   // GBK_TO_UNICODE[6993] := 16#6436;
   // GBK_TO_UNICODE[6994] := 16#938D;
   // GBK_TO_UNICODE[6995] := 16#6437;
   // GBK_TO_UNICODE[6996] := 16#938E;
   // GBK_TO_UNICODE[6997] := 16#6438;
   // GBK_TO_UNICODE[6998] := 16#938F;
   // GBK_TO_UNICODE[6999] := 16#6439;
   // GBK_TO_UNICODE[7000] := 16#9390;
   // GBK_TO_UNICODE[7001] := 16#643B;
   // GBK_TO_UNICODE[7002] := 16#9391;
   // GBK_TO_UNICODE[7003] := 16#643C;
   // GBK_TO_UNICODE[7004] := 16#9392;
   // GBK_TO_UNICODE[7005] := 16#643E;
   // GBK_TO_UNICODE[7006] := 16#9393;
   // GBK_TO_UNICODE[7007] := 16#6440;
   // GBK_TO_UNICODE[7008] := 16#9394;
   // GBK_TO_UNICODE[7009] := 16#6442;
   // GBK_TO_UNICODE[7010] := 16#9395;
   // GBK_TO_UNICODE[7011] := 16#6443;
   // GBK_TO_UNICODE[7012] := 16#9396;
   // GBK_TO_UNICODE[7013] := 16#6449;
   // GBK_TO_UNICODE[7014] := 16#9397;
   // GBK_TO_UNICODE[7015] := 16#644B;
   // GBK_TO_UNICODE[7016] := 16#9398;
   // GBK_TO_UNICODE[7017] := 16#644C;
   // GBK_TO_UNICODE[7018] := 16#9399;
   // GBK_TO_UNICODE[7019] := 16#644D;
   // GBK_TO_UNICODE[7020] := 16#939A;
   // GBK_TO_UNICODE[7021] := 16#644E;
   // GBK_TO_UNICODE[7022] := 16#939B;
   // GBK_TO_UNICODE[7023] := 16#644F;
   // GBK_TO_UNICODE[7024] := 16#939C;
   // GBK_TO_UNICODE[7025] := 16#6450;
   // GBK_TO_UNICODE[7026] := 16#939D;
   // GBK_TO_UNICODE[7027] := 16#6451;
   // GBK_TO_UNICODE[7028] := 16#939E;
   // GBK_TO_UNICODE[7029] := 16#6453;
   // GBK_TO_UNICODE[7030] := 16#939F;
   // GBK_TO_UNICODE[7031] := 16#6455;
   // GBK_TO_UNICODE[7032] := 16#93A0;
   // GBK_TO_UNICODE[7033] := 16#6456;
   // GBK_TO_UNICODE[7034] := 16#93A1;
   // GBK_TO_UNICODE[7035] := 16#6457;
   // GBK_TO_UNICODE[7036] := 16#93A2;
   // GBK_TO_UNICODE[7037] := 16#6459;
   // GBK_TO_UNICODE[7038] := 16#93A3;
   // GBK_TO_UNICODE[7039] := 16#645A;
   // GBK_TO_UNICODE[7040] := 16#93A4;
   // GBK_TO_UNICODE[7041] := 16#645B;
   // GBK_TO_UNICODE[7042] := 16#93A5;
   // GBK_TO_UNICODE[7043] := 16#645C;
   // GBK_TO_UNICODE[7044] := 16#93A6;
   // GBK_TO_UNICODE[7045] := 16#645D;
   // GBK_TO_UNICODE[7046] := 16#93A7;
   // GBK_TO_UNICODE[7047] := 16#645F;
   // GBK_TO_UNICODE[7048] := 16#93A8;
   // GBK_TO_UNICODE[7049] := 16#6460;
   // GBK_TO_UNICODE[7050] := 16#93A9;
   // GBK_TO_UNICODE[7051] := 16#6461;
   // GBK_TO_UNICODE[7052] := 16#93AA;
   // GBK_TO_UNICODE[7053] := 16#6462;
   // GBK_TO_UNICODE[7054] := 16#93AB;
   // GBK_TO_UNICODE[7055] := 16#6463;
   // GBK_TO_UNICODE[7056] := 16#93AC;
   // GBK_TO_UNICODE[7057] := 16#6464;
   // GBK_TO_UNICODE[7058] := 16#93AD;
   // GBK_TO_UNICODE[7059] := 16#6465;
   // GBK_TO_UNICODE[7060] := 16#93AE;
   // GBK_TO_UNICODE[7061] := 16#6466;
   // GBK_TO_UNICODE[7062] := 16#93AF;
   // GBK_TO_UNICODE[7063] := 16#6468;
   // GBK_TO_UNICODE[7064] := 16#93B0;
   // GBK_TO_UNICODE[7065] := 16#646A;
   // GBK_TO_UNICODE[7066] := 16#93B1;
   // GBK_TO_UNICODE[7067] := 16#646B;
   // GBK_TO_UNICODE[7068] := 16#93B2;
   // GBK_TO_UNICODE[7069] := 16#646C;
   // GBK_TO_UNICODE[7070] := 16#93B3;
   // GBK_TO_UNICODE[7071] := 16#646E;
   // GBK_TO_UNICODE[7072] := 16#93B4;
   // GBK_TO_UNICODE[7073] := 16#646F;
   // GBK_TO_UNICODE[7074] := 16#93B5;
   // GBK_TO_UNICODE[7075] := 16#6470;
   // GBK_TO_UNICODE[7076] := 16#93B6;
   // GBK_TO_UNICODE[7077] := 16#6471;
   // GBK_TO_UNICODE[7078] := 16#93B7;
   // GBK_TO_UNICODE[7079] := 16#6472;
   // GBK_TO_UNICODE[7080] := 16#93B8;
   // GBK_TO_UNICODE[7081] := 16#6473;
   // GBK_TO_UNICODE[7082] := 16#93B9;
   // GBK_TO_UNICODE[7083] := 16#6474;
   // GBK_TO_UNICODE[7084] := 16#93BA;
   // GBK_TO_UNICODE[7085] := 16#6475;
   // GBK_TO_UNICODE[7086] := 16#93BB;
   // GBK_TO_UNICODE[7087] := 16#6476;
   // GBK_TO_UNICODE[7088] := 16#93BC;
   // GBK_TO_UNICODE[7089] := 16#6477;
   // GBK_TO_UNICODE[7090] := 16#93BD;
   // GBK_TO_UNICODE[7091] := 16#647B;
   // GBK_TO_UNICODE[7092] := 16#93BE;
   // GBK_TO_UNICODE[7093] := 16#647C;
   // GBK_TO_UNICODE[7094] := 16#93BF;
   // GBK_TO_UNICODE[7095] := 16#647D;
   // GBK_TO_UNICODE[7096] := 16#93C0;
   // GBK_TO_UNICODE[7097] := 16#647E;
   // GBK_TO_UNICODE[7098] := 16#93C1;
   // GBK_TO_UNICODE[7099] := 16#647F;
   // GBK_TO_UNICODE[7100] := 16#93C2;
   // GBK_TO_UNICODE[7101] := 16#6480;
   // GBK_TO_UNICODE[7102] := 16#93C3;
   // GBK_TO_UNICODE[7103] := 16#6481;
   // GBK_TO_UNICODE[7104] := 16#93C4;
   // GBK_TO_UNICODE[7105] := 16#6483;
   // GBK_TO_UNICODE[7106] := 16#93C5;
   // GBK_TO_UNICODE[7107] := 16#6486;
   // GBK_TO_UNICODE[7108] := 16#93C6;
   // GBK_TO_UNICODE[7109] := 16#6488;
   // GBK_TO_UNICODE[7110] := 16#93C7;
   // GBK_TO_UNICODE[7111] := 16#6489;
   // GBK_TO_UNICODE[7112] := 16#93C8;
   // GBK_TO_UNICODE[7113] := 16#648A;
   // GBK_TO_UNICODE[7114] := 16#93C9;
   // GBK_TO_UNICODE[7115] := 16#648B;
   // GBK_TO_UNICODE[7116] := 16#93CA;
   // GBK_TO_UNICODE[7117] := 16#648C;
   // GBK_TO_UNICODE[7118] := 16#93CB;
   // GBK_TO_UNICODE[7119] := 16#648D;
   // GBK_TO_UNICODE[7120] := 16#93CC;
   // GBK_TO_UNICODE[7121] := 16#648E;
   // GBK_TO_UNICODE[7122] := 16#93CD;
   // GBK_TO_UNICODE[7123] := 16#648F;
   // GBK_TO_UNICODE[7124] := 16#93CE;
   // GBK_TO_UNICODE[7125] := 16#6490;
   // GBK_TO_UNICODE[7126] := 16#93CF;
   // GBK_TO_UNICODE[7127] := 16#6493;
   // GBK_TO_UNICODE[7128] := 16#93D0;
   // GBK_TO_UNICODE[7129] := 16#6494;
   // GBK_TO_UNICODE[7130] := 16#93D1;
   // GBK_TO_UNICODE[7131] := 16#6497;
   // GBK_TO_UNICODE[7132] := 16#93D2;
   // GBK_TO_UNICODE[7133] := 16#6498;
   // GBK_TO_UNICODE[7134] := 16#93D3;
   // GBK_TO_UNICODE[7135] := 16#649A;
   // GBK_TO_UNICODE[7136] := 16#93D4;
   // GBK_TO_UNICODE[7137] := 16#649B;
   // GBK_TO_UNICODE[7138] := 16#93D5;
   // GBK_TO_UNICODE[7139] := 16#649C;
   // GBK_TO_UNICODE[7140] := 16#93D6;
   // GBK_TO_UNICODE[7141] := 16#649D;
   // GBK_TO_UNICODE[7142] := 16#93D7;
   // GBK_TO_UNICODE[7143] := 16#649F;
   // GBK_TO_UNICODE[7144] := 16#93D8;
   // GBK_TO_UNICODE[7145] := 16#64A0;
   // GBK_TO_UNICODE[7146] := 16#93D9;
   // GBK_TO_UNICODE[7147] := 16#64A1;
   // GBK_TO_UNICODE[7148] := 16#93DA;
   // GBK_TO_UNICODE[7149] := 16#64A2;
   // GBK_TO_UNICODE[7150] := 16#93DB;
   // GBK_TO_UNICODE[7151] := 16#64A3;
   // GBK_TO_UNICODE[7152] := 16#93DC;
   // GBK_TO_UNICODE[7153] := 16#64A5;
   // GBK_TO_UNICODE[7154] := 16#93DD;
   // GBK_TO_UNICODE[7155] := 16#64A6;
   // GBK_TO_UNICODE[7156] := 16#93DE;
   // GBK_TO_UNICODE[7157] := 16#64A7;
   // GBK_TO_UNICODE[7158] := 16#93DF;
   // GBK_TO_UNICODE[7159] := 16#64A8;
   // GBK_TO_UNICODE[7160] := 16#93E0;
   // GBK_TO_UNICODE[7161] := 16#64AA;
   // GBK_TO_UNICODE[7162] := 16#93E1;
   // GBK_TO_UNICODE[7163] := 16#64AB;
   // GBK_TO_UNICODE[7164] := 16#93E2;
   // GBK_TO_UNICODE[7165] := 16#64AF;
   // GBK_TO_UNICODE[7166] := 16#93E3;
   // GBK_TO_UNICODE[7167] := 16#64B1;
   // GBK_TO_UNICODE[7168] := 16#93E4;
   // GBK_TO_UNICODE[7169] := 16#64B2;
   // GBK_TO_UNICODE[7170] := 16#93E5;
   // GBK_TO_UNICODE[7171] := 16#64B3;
   // GBK_TO_UNICODE[7172] := 16#93E6;
   // GBK_TO_UNICODE[7173] := 16#64B4;
   // GBK_TO_UNICODE[7174] := 16#93E7;
   // GBK_TO_UNICODE[7175] := 16#64B6;
   // GBK_TO_UNICODE[7176] := 16#93E8;
   // GBK_TO_UNICODE[7177] := 16#64B9;
   // GBK_TO_UNICODE[7178] := 16#93E9;
   // GBK_TO_UNICODE[7179] := 16#64BB;
   // GBK_TO_UNICODE[7180] := 16#93EA;
   // GBK_TO_UNICODE[7181] := 16#64BD;
   // GBK_TO_UNICODE[7182] := 16#93EB;
   // GBK_TO_UNICODE[7183] := 16#64BE;
   // GBK_TO_UNICODE[7184] := 16#93EC;
   // GBK_TO_UNICODE[7185] := 16#64BF;
   // GBK_TO_UNICODE[7186] := 16#93ED;
   // GBK_TO_UNICODE[7187] := 16#64C1;
   // GBK_TO_UNICODE[7188] := 16#93EE;
   // GBK_TO_UNICODE[7189] := 16#64C3;
   // GBK_TO_UNICODE[7190] := 16#93EF;
   // GBK_TO_UNICODE[7191] := 16#64C4;
   // GBK_TO_UNICODE[7192] := 16#93F0;
   // GBK_TO_UNICODE[7193] := 16#64C6;
   // GBK_TO_UNICODE[7194] := 16#93F1;
   // GBK_TO_UNICODE[7195] := 16#64C7;
   // GBK_TO_UNICODE[7196] := 16#93F2;
   // GBK_TO_UNICODE[7197] := 16#64C8;
   // GBK_TO_UNICODE[7198] := 16#93F3;
   // GBK_TO_UNICODE[7199] := 16#64C9;
   // GBK_TO_UNICODE[7200] := 16#93F4;
   // GBK_TO_UNICODE[7201] := 16#64CA;
   // GBK_TO_UNICODE[7202] := 16#93F5;
   // GBK_TO_UNICODE[7203] := 16#64CB;
   // GBK_TO_UNICODE[7204] := 16#93F6;
   // GBK_TO_UNICODE[7205] := 16#64CC;
   // GBK_TO_UNICODE[7206] := 16#93F7;
   // GBK_TO_UNICODE[7207] := 16#64CF;
   // GBK_TO_UNICODE[7208] := 16#93F8;
   // GBK_TO_UNICODE[7209] := 16#64D1;
   // GBK_TO_UNICODE[7210] := 16#93F9;
   // GBK_TO_UNICODE[7211] := 16#64D3;
   // GBK_TO_UNICODE[7212] := 16#93FA;
   // GBK_TO_UNICODE[7213] := 16#64D4;
   // GBK_TO_UNICODE[7214] := 16#93FB;
   // GBK_TO_UNICODE[7215] := 16#64D5;
   // GBK_TO_UNICODE[7216] := 16#93FC;
   // GBK_TO_UNICODE[7217] := 16#64D6;
   // GBK_TO_UNICODE[7218] := 16#93FD;
   // GBK_TO_UNICODE[7219] := 16#64D9;
   // GBK_TO_UNICODE[7220] := 16#93FE;
   // GBK_TO_UNICODE[7221] := 16#64DA;
   // GBK_TO_UNICODE[7222] := 16#9440;
   // GBK_TO_UNICODE[7223] := 16#64DB;
   // GBK_TO_UNICODE[7224] := 16#9441;
   // GBK_TO_UNICODE[7225] := 16#64DC;
   // GBK_TO_UNICODE[7226] := 16#9442;
   // GBK_TO_UNICODE[7227] := 16#64DD;
   // GBK_TO_UNICODE[7228] := 16#9443;
   // GBK_TO_UNICODE[7229] := 16#64DF;
   // GBK_TO_UNICODE[7230] := 16#9444;
   // GBK_TO_UNICODE[7231] := 16#64E0;
   // GBK_TO_UNICODE[7232] := 16#9445;
   // GBK_TO_UNICODE[7233] := 16#64E1;
   // GBK_TO_UNICODE[7234] := 16#9446;
   // GBK_TO_UNICODE[7235] := 16#64E3;
   // GBK_TO_UNICODE[7236] := 16#9447;
   // GBK_TO_UNICODE[7237] := 16#64E5;
   // GBK_TO_UNICODE[7238] := 16#9448;
   // GBK_TO_UNICODE[7239] := 16#64E7;
   // GBK_TO_UNICODE[7240] := 16#9449;
   // GBK_TO_UNICODE[7241] := 16#64E8;
   // GBK_TO_UNICODE[7242] := 16#944A;
   // GBK_TO_UNICODE[7243] := 16#64E9;
   // GBK_TO_UNICODE[7244] := 16#944B;
   // GBK_TO_UNICODE[7245] := 16#64EA;
   // GBK_TO_UNICODE[7246] := 16#944C;
   // GBK_TO_UNICODE[7247] := 16#64EB;
   // GBK_TO_UNICODE[7248] := 16#944D;
   // GBK_TO_UNICODE[7249] := 16#64EC;
   // GBK_TO_UNICODE[7250] := 16#944E;
   // GBK_TO_UNICODE[7251] := 16#64ED;
   // GBK_TO_UNICODE[7252] := 16#944F;
   // GBK_TO_UNICODE[7253] := 16#64EE;
   // GBK_TO_UNICODE[7254] := 16#9450;
   // GBK_TO_UNICODE[7255] := 16#64EF;
   // GBK_TO_UNICODE[7256] := 16#9451;
   // GBK_TO_UNICODE[7257] := 16#64F0;
   // GBK_TO_UNICODE[7258] := 16#9452;
   // GBK_TO_UNICODE[7259] := 16#64F1;
   // GBK_TO_UNICODE[7260] := 16#9453;
   // GBK_TO_UNICODE[7261] := 16#64F2;
   // GBK_TO_UNICODE[7262] := 16#9454;
   // GBK_TO_UNICODE[7263] := 16#64F3;
   // GBK_TO_UNICODE[7264] := 16#9455;
   // GBK_TO_UNICODE[7265] := 16#64F4;
   // GBK_TO_UNICODE[7266] := 16#9456;
   // GBK_TO_UNICODE[7267] := 16#64F5;
   // GBK_TO_UNICODE[7268] := 16#9457;
   // GBK_TO_UNICODE[7269] := 16#64F6;
   // GBK_TO_UNICODE[7270] := 16#9458;
   // GBK_TO_UNICODE[7271] := 16#64F7;
   // GBK_TO_UNICODE[7272] := 16#9459;
   // GBK_TO_UNICODE[7273] := 16#64F8;
   // GBK_TO_UNICODE[7274] := 16#945A;
   // GBK_TO_UNICODE[7275] := 16#64F9;
   // GBK_TO_UNICODE[7276] := 16#945B;
   // GBK_TO_UNICODE[7277] := 16#64FA;
   // GBK_TO_UNICODE[7278] := 16#945C;
   // GBK_TO_UNICODE[7279] := 16#64FB;
   // GBK_TO_UNICODE[7280] := 16#945D;
   // GBK_TO_UNICODE[7281] := 16#64FC;
   // GBK_TO_UNICODE[7282] := 16#945E;
   // GBK_TO_UNICODE[7283] := 16#64FD;
   // GBK_TO_UNICODE[7284] := 16#945F;
   // GBK_TO_UNICODE[7285] := 16#64FE;
   // GBK_TO_UNICODE[7286] := 16#9460;
   // GBK_TO_UNICODE[7287] := 16#64FF;
   // GBK_TO_UNICODE[7288] := 16#9461;
   // GBK_TO_UNICODE[7289] := 16#6501;
   // GBK_TO_UNICODE[7290] := 16#9462;
   // GBK_TO_UNICODE[7291] := 16#6502;
   // GBK_TO_UNICODE[7292] := 16#9463;
   // GBK_TO_UNICODE[7293] := 16#6503;
   // GBK_TO_UNICODE[7294] := 16#9464;
   // GBK_TO_UNICODE[7295] := 16#6504;
   // GBK_TO_UNICODE[7296] := 16#9465;
   // GBK_TO_UNICODE[7297] := 16#6505;
   // GBK_TO_UNICODE[7298] := 16#9466;
   // GBK_TO_UNICODE[7299] := 16#6506;
   // GBK_TO_UNICODE[7300] := 16#9467;
   // GBK_TO_UNICODE[7301] := 16#6507;
   // GBK_TO_UNICODE[7302] := 16#9468;
   // GBK_TO_UNICODE[7303] := 16#6508;
   // GBK_TO_UNICODE[7304] := 16#9469;
   // GBK_TO_UNICODE[7305] := 16#650A;
   // GBK_TO_UNICODE[7306] := 16#946A;
   // GBK_TO_UNICODE[7307] := 16#650B;
   // GBK_TO_UNICODE[7308] := 16#946B;
   // GBK_TO_UNICODE[7309] := 16#650C;
   // GBK_TO_UNICODE[7310] := 16#946C;
   // GBK_TO_UNICODE[7311] := 16#650D;
   // GBK_TO_UNICODE[7312] := 16#946D;
   // GBK_TO_UNICODE[7313] := 16#650E;
   // GBK_TO_UNICODE[7314] := 16#946E;
   // GBK_TO_UNICODE[7315] := 16#650F;
   // GBK_TO_UNICODE[7316] := 16#946F;
   // GBK_TO_UNICODE[7317] := 16#6510;
   // GBK_TO_UNICODE[7318] := 16#9470;
   // GBK_TO_UNICODE[7319] := 16#6511;
   // GBK_TO_UNICODE[7320] := 16#9471;
   // GBK_TO_UNICODE[7321] := 16#6513;
   // GBK_TO_UNICODE[7322] := 16#9472;
   // GBK_TO_UNICODE[7323] := 16#6514;
   // GBK_TO_UNICODE[7324] := 16#9473;
   // GBK_TO_UNICODE[7325] := 16#6515;
   // GBK_TO_UNICODE[7326] := 16#9474;
   // GBK_TO_UNICODE[7327] := 16#6516;
   // GBK_TO_UNICODE[7328] := 16#9475;
   // GBK_TO_UNICODE[7329] := 16#6517;
   // GBK_TO_UNICODE[7330] := 16#9476;
   // GBK_TO_UNICODE[7331] := 16#6519;
   // GBK_TO_UNICODE[7332] := 16#9477;
   // GBK_TO_UNICODE[7333] := 16#651A;
   // GBK_TO_UNICODE[7334] := 16#9478;
   // GBK_TO_UNICODE[7335] := 16#651B;
   // GBK_TO_UNICODE[7336] := 16#9479;
   // GBK_TO_UNICODE[7337] := 16#651C;
   // GBK_TO_UNICODE[7338] := 16#947A;
   // GBK_TO_UNICODE[7339] := 16#651D;
   // GBK_TO_UNICODE[7340] := 16#947B;
   // GBK_TO_UNICODE[7341] := 16#651E;
   // GBK_TO_UNICODE[7342] := 16#947C;
   // GBK_TO_UNICODE[7343] := 16#651F;
   // GBK_TO_UNICODE[7344] := 16#947D;
   // GBK_TO_UNICODE[7345] := 16#6520;
   // GBK_TO_UNICODE[7346] := 16#947E;
   // GBK_TO_UNICODE[7347] := 16#6521;
   // GBK_TO_UNICODE[7348] := 16#9480;
   // GBK_TO_UNICODE[7349] := 16#6522;
   // GBK_TO_UNICODE[7350] := 16#9481;
   // GBK_TO_UNICODE[7351] := 16#6523;
   // GBK_TO_UNICODE[7352] := 16#9482;
   // GBK_TO_UNICODE[7353] := 16#6524;
   // GBK_TO_UNICODE[7354] := 16#9483;
   // GBK_TO_UNICODE[7355] := 16#6526;
   // GBK_TO_UNICODE[7356] := 16#9484;
   // GBK_TO_UNICODE[7357] := 16#6527;
   // GBK_TO_UNICODE[7358] := 16#9485;
   // GBK_TO_UNICODE[7359] := 16#6528;
   // GBK_TO_UNICODE[7360] := 16#9486;
   // GBK_TO_UNICODE[7361] := 16#6529;
   // GBK_TO_UNICODE[7362] := 16#9487;
   // GBK_TO_UNICODE[7363] := 16#652A;
   // GBK_TO_UNICODE[7364] := 16#9488;
   // GBK_TO_UNICODE[7365] := 16#652C;
   // GBK_TO_UNICODE[7366] := 16#9489;
   // GBK_TO_UNICODE[7367] := 16#652D;
   // GBK_TO_UNICODE[7368] := 16#948A;
   // GBK_TO_UNICODE[7369] := 16#6530;
   // GBK_TO_UNICODE[7370] := 16#948B;
   // GBK_TO_UNICODE[7371] := 16#6531;
   // GBK_TO_UNICODE[7372] := 16#948C;
   // GBK_TO_UNICODE[7373] := 16#6532;
   // GBK_TO_UNICODE[7374] := 16#948D;
   // GBK_TO_UNICODE[7375] := 16#6533;
   // GBK_TO_UNICODE[7376] := 16#948E;
   // GBK_TO_UNICODE[7377] := 16#6537;
   // GBK_TO_UNICODE[7378] := 16#948F;
   // GBK_TO_UNICODE[7379] := 16#653A;
   // GBK_TO_UNICODE[7380] := 16#9490;
   // GBK_TO_UNICODE[7381] := 16#653C;
   // GBK_TO_UNICODE[7382] := 16#9491;
   // GBK_TO_UNICODE[7383] := 16#653D;
   // GBK_TO_UNICODE[7384] := 16#9492;
   // GBK_TO_UNICODE[7385] := 16#6540;
   // GBK_TO_UNICODE[7386] := 16#9493;
   // GBK_TO_UNICODE[7387] := 16#6541;
   // GBK_TO_UNICODE[7388] := 16#9494;
   // GBK_TO_UNICODE[7389] := 16#6542;
   // GBK_TO_UNICODE[7390] := 16#9495;
   // GBK_TO_UNICODE[7391] := 16#6543;
   // GBK_TO_UNICODE[7392] := 16#9496;
   // GBK_TO_UNICODE[7393] := 16#6544;
   // GBK_TO_UNICODE[7394] := 16#9497;
   // GBK_TO_UNICODE[7395] := 16#6546;
   // GBK_TO_UNICODE[7396] := 16#9498;
   // GBK_TO_UNICODE[7397] := 16#6547;
   // GBK_TO_UNICODE[7398] := 16#9499;
   // GBK_TO_UNICODE[7399] := 16#654A;
   // GBK_TO_UNICODE[7400] := 16#949A;
   // GBK_TO_UNICODE[7401] := 16#654B;
   // GBK_TO_UNICODE[7402] := 16#949B;
   // GBK_TO_UNICODE[7403] := 16#654D;
   // GBK_TO_UNICODE[7404] := 16#949C;
   // GBK_TO_UNICODE[7405] := 16#654E;
   // GBK_TO_UNICODE[7406] := 16#949D;
   // GBK_TO_UNICODE[7407] := 16#6550;
   // GBK_TO_UNICODE[7408] := 16#949E;
   // GBK_TO_UNICODE[7409] := 16#6552;
   // GBK_TO_UNICODE[7410] := 16#949F;
   // GBK_TO_UNICODE[7411] := 16#6553;
   // GBK_TO_UNICODE[7412] := 16#94A0;
   // GBK_TO_UNICODE[7413] := 16#6554;
   // GBK_TO_UNICODE[7414] := 16#94A1;
   // GBK_TO_UNICODE[7415] := 16#6557;
   // GBK_TO_UNICODE[7416] := 16#94A2;
   // GBK_TO_UNICODE[7417] := 16#6558;
   // GBK_TO_UNICODE[7418] := 16#94A3;
   // GBK_TO_UNICODE[7419] := 16#655A;
   // GBK_TO_UNICODE[7420] := 16#94A4;
   // GBK_TO_UNICODE[7421] := 16#655C;
   // GBK_TO_UNICODE[7422] := 16#94A5;
   // GBK_TO_UNICODE[7423] := 16#655F;
   // GBK_TO_UNICODE[7424] := 16#94A6;
   // GBK_TO_UNICODE[7425] := 16#6560;
   // GBK_TO_UNICODE[7426] := 16#94A7;
   // GBK_TO_UNICODE[7427] := 16#6561;
   // GBK_TO_UNICODE[7428] := 16#94A8;
   // GBK_TO_UNICODE[7429] := 16#6564;
   // GBK_TO_UNICODE[7430] := 16#94A9;
   // GBK_TO_UNICODE[7431] := 16#6565;
   // GBK_TO_UNICODE[7432] := 16#94AA;
   // GBK_TO_UNICODE[7433] := 16#6567;
   // GBK_TO_UNICODE[7434] := 16#94AB;
   // GBK_TO_UNICODE[7435] := 16#6568;
   // GBK_TO_UNICODE[7436] := 16#94AC;
   // GBK_TO_UNICODE[7437] := 16#6569;
   // GBK_TO_UNICODE[7438] := 16#94AD;
   // GBK_TO_UNICODE[7439] := 16#656A;
   // GBK_TO_UNICODE[7440] := 16#94AE;
   // GBK_TO_UNICODE[7441] := 16#656D;
   // GBK_TO_UNICODE[7442] := 16#94AF;
   // GBK_TO_UNICODE[7443] := 16#656E;
   // GBK_TO_UNICODE[7444] := 16#94B0;
   // GBK_TO_UNICODE[7445] := 16#656F;
   // GBK_TO_UNICODE[7446] := 16#94B1;
   // GBK_TO_UNICODE[7447] := 16#6571;
   // GBK_TO_UNICODE[7448] := 16#94B2;
   // GBK_TO_UNICODE[7449] := 16#6573;
   // GBK_TO_UNICODE[7450] := 16#94B3;
   // GBK_TO_UNICODE[7451] := 16#6575;
   // GBK_TO_UNICODE[7452] := 16#94B4;
   // GBK_TO_UNICODE[7453] := 16#6576;
   // GBK_TO_UNICODE[7454] := 16#94B5;
   // GBK_TO_UNICODE[7455] := 16#6578;
   // GBK_TO_UNICODE[7456] := 16#94B6;
   // GBK_TO_UNICODE[7457] := 16#6579;
   // GBK_TO_UNICODE[7458] := 16#94B7;
   // GBK_TO_UNICODE[7459] := 16#657A;
   // GBK_TO_UNICODE[7460] := 16#94B8;
   // GBK_TO_UNICODE[7461] := 16#657B;
   // GBK_TO_UNICODE[7462] := 16#94B9;
   // GBK_TO_UNICODE[7463] := 16#657C;
   // GBK_TO_UNICODE[7464] := 16#94BA;
   // GBK_TO_UNICODE[7465] := 16#657D;
   // GBK_TO_UNICODE[7466] := 16#94BB;
   // GBK_TO_UNICODE[7467] := 16#657E;
   // GBK_TO_UNICODE[7468] := 16#94BC;
   // GBK_TO_UNICODE[7469] := 16#657F;
   // GBK_TO_UNICODE[7470] := 16#94BD;
   // GBK_TO_UNICODE[7471] := 16#6580;
   // GBK_TO_UNICODE[7472] := 16#94BE;
   // GBK_TO_UNICODE[7473] := 16#6581;
   // GBK_TO_UNICODE[7474] := 16#94BF;
   // GBK_TO_UNICODE[7475] := 16#6582;
   // GBK_TO_UNICODE[7476] := 16#94C0;
   // GBK_TO_UNICODE[7477] := 16#6583;
   // GBK_TO_UNICODE[7478] := 16#94C1;
   // GBK_TO_UNICODE[7479] := 16#6584;
   // GBK_TO_UNICODE[7480] := 16#94C2;
   // GBK_TO_UNICODE[7481] := 16#6585;
   // GBK_TO_UNICODE[7482] := 16#94C3;
   // GBK_TO_UNICODE[7483] := 16#6586;
   // GBK_TO_UNICODE[7484] := 16#94C4;
   // GBK_TO_UNICODE[7485] := 16#6588;
   // GBK_TO_UNICODE[7486] := 16#94C5;
   // GBK_TO_UNICODE[7487] := 16#6589;
   // GBK_TO_UNICODE[7488] := 16#94C6;
   // GBK_TO_UNICODE[7489] := 16#658A;
   // GBK_TO_UNICODE[7490] := 16#94C7;
   // GBK_TO_UNICODE[7491] := 16#658D;
   // GBK_TO_UNICODE[7492] := 16#94C8;
   // GBK_TO_UNICODE[7493] := 16#658E;
   // GBK_TO_UNICODE[7494] := 16#94C9;
   // GBK_TO_UNICODE[7495] := 16#658F;
   // GBK_TO_UNICODE[7496] := 16#94CA;
   // GBK_TO_UNICODE[7497] := 16#6592;
   // GBK_TO_UNICODE[7498] := 16#94CB;
   // GBK_TO_UNICODE[7499] := 16#6594;
   // GBK_TO_UNICODE[7500] := 16#94CC;
   // GBK_TO_UNICODE[7501] := 16#6595;
   // GBK_TO_UNICODE[7502] := 16#94CD;
   // GBK_TO_UNICODE[7503] := 16#6596;
   // GBK_TO_UNICODE[7504] := 16#94CE;
   // GBK_TO_UNICODE[7505] := 16#6598;
   // GBK_TO_UNICODE[7506] := 16#94CF;
   // GBK_TO_UNICODE[7507] := 16#659A;
   // GBK_TO_UNICODE[7508] := 16#94D0;
   // GBK_TO_UNICODE[7509] := 16#659D;
   // GBK_TO_UNICODE[7510] := 16#94D1;
   // GBK_TO_UNICODE[7511] := 16#659E;
   // GBK_TO_UNICODE[7512] := 16#94D2;
   // GBK_TO_UNICODE[7513] := 16#65A0;
   // GBK_TO_UNICODE[7514] := 16#94D3;
   // GBK_TO_UNICODE[7515] := 16#65A2;
   // GBK_TO_UNICODE[7516] := 16#94D4;
   // GBK_TO_UNICODE[7517] := 16#65A3;
   // GBK_TO_UNICODE[7518] := 16#94D5;
   // GBK_TO_UNICODE[7519] := 16#65A6;
   // GBK_TO_UNICODE[7520] := 16#94D6;
   // GBK_TO_UNICODE[7521] := 16#65A8;
   // GBK_TO_UNICODE[7522] := 16#94D7;
   // GBK_TO_UNICODE[7523] := 16#65AA;
   // GBK_TO_UNICODE[7524] := 16#94D8;
   // GBK_TO_UNICODE[7525] := 16#65AC;
   // GBK_TO_UNICODE[7526] := 16#94D9;
   // GBK_TO_UNICODE[7527] := 16#65AE;
   // GBK_TO_UNICODE[7528] := 16#94DA;
   // GBK_TO_UNICODE[7529] := 16#65B1;
   // GBK_TO_UNICODE[7530] := 16#94DB;
   // GBK_TO_UNICODE[7531] := 16#65B2;
   // GBK_TO_UNICODE[7532] := 16#94DC;
   // GBK_TO_UNICODE[7533] := 16#65B3;
   // GBK_TO_UNICODE[7534] := 16#94DD;
   // GBK_TO_UNICODE[7535] := 16#65B4;
   // GBK_TO_UNICODE[7536] := 16#94DE;
   // GBK_TO_UNICODE[7537] := 16#65B5;
   // GBK_TO_UNICODE[7538] := 16#94DF;
   // GBK_TO_UNICODE[7539] := 16#65B6;
   // GBK_TO_UNICODE[7540] := 16#94E0;
   // GBK_TO_UNICODE[7541] := 16#65B7;
   // GBK_TO_UNICODE[7542] := 16#94E1;
   // GBK_TO_UNICODE[7543] := 16#65B8;
   // GBK_TO_UNICODE[7544] := 16#94E2;
   // GBK_TO_UNICODE[7545] := 16#65BA;
   // GBK_TO_UNICODE[7546] := 16#94E3;
   // GBK_TO_UNICODE[7547] := 16#65BB;
   // GBK_TO_UNICODE[7548] := 16#94E4;
   // GBK_TO_UNICODE[7549] := 16#65BE;
   // GBK_TO_UNICODE[7550] := 16#94E5;
   // GBK_TO_UNICODE[7551] := 16#65BF;
   // GBK_TO_UNICODE[7552] := 16#94E6;
   // GBK_TO_UNICODE[7553] := 16#65C0;
   // GBK_TO_UNICODE[7554] := 16#94E7;
   // GBK_TO_UNICODE[7555] := 16#65C2;
   // GBK_TO_UNICODE[7556] := 16#94E8;
   // GBK_TO_UNICODE[7557] := 16#65C7;
   // GBK_TO_UNICODE[7558] := 16#94E9;
   // GBK_TO_UNICODE[7559] := 16#65C8;
   // GBK_TO_UNICODE[7560] := 16#94EA;
   // GBK_TO_UNICODE[7561] := 16#65C9;
   // GBK_TO_UNICODE[7562] := 16#94EB;
   // GBK_TO_UNICODE[7563] := 16#65CA;
   // GBK_TO_UNICODE[7564] := 16#94EC;
   // GBK_TO_UNICODE[7565] := 16#65CD;
   // GBK_TO_UNICODE[7566] := 16#94ED;
   // GBK_TO_UNICODE[7567] := 16#65D0;
   // GBK_TO_UNICODE[7568] := 16#94EE;
   // GBK_TO_UNICODE[7569] := 16#65D1;
   // GBK_TO_UNICODE[7570] := 16#94EF;
   // GBK_TO_UNICODE[7571] := 16#65D3;
   // GBK_TO_UNICODE[7572] := 16#94F0;
   // GBK_TO_UNICODE[7573] := 16#65D4;
   // GBK_TO_UNICODE[7574] := 16#94F1;
   // GBK_TO_UNICODE[7575] := 16#65D5;
   // GBK_TO_UNICODE[7576] := 16#94F2;
   // GBK_TO_UNICODE[7577] := 16#65D8;
   // GBK_TO_UNICODE[7578] := 16#94F3;
   // GBK_TO_UNICODE[7579] := 16#65D9;
   // GBK_TO_UNICODE[7580] := 16#94F4;
   // GBK_TO_UNICODE[7581] := 16#65DA;
   // GBK_TO_UNICODE[7582] := 16#94F5;
   // GBK_TO_UNICODE[7583] := 16#65DB;
   // GBK_TO_UNICODE[7584] := 16#94F6;
   // GBK_TO_UNICODE[7585] := 16#65DC;
   // GBK_TO_UNICODE[7586] := 16#94F7;
   // GBK_TO_UNICODE[7587] := 16#65DD;
   // GBK_TO_UNICODE[7588] := 16#94F8;
   // GBK_TO_UNICODE[7589] := 16#65DE;
   // GBK_TO_UNICODE[7590] := 16#94F9;
   // GBK_TO_UNICODE[7591] := 16#65DF;
   // GBK_TO_UNICODE[7592] := 16#94FA;
   // GBK_TO_UNICODE[7593] := 16#65E1;
   // GBK_TO_UNICODE[7594] := 16#94FB;
   // GBK_TO_UNICODE[7595] := 16#65E3;
   // GBK_TO_UNICODE[7596] := 16#94FC;
   // GBK_TO_UNICODE[7597] := 16#65E4;
   // GBK_TO_UNICODE[7598] := 16#94FD;
   // GBK_TO_UNICODE[7599] := 16#65EA;
   // GBK_TO_UNICODE[7600] := 16#94FE;
   // GBK_TO_UNICODE[7601] := 16#65EB;
   // GBK_TO_UNICODE[7602] := 16#9540;
   // GBK_TO_UNICODE[7603] := 16#65F2;
   // GBK_TO_UNICODE[7604] := 16#9541;
   // GBK_TO_UNICODE[7605] := 16#65F3;
   // GBK_TO_UNICODE[7606] := 16#9542;
   // GBK_TO_UNICODE[7607] := 16#65F4;
   // GBK_TO_UNICODE[7608] := 16#9543;
   // GBK_TO_UNICODE[7609] := 16#65F5;
   // GBK_TO_UNICODE[7610] := 16#9544;
   // GBK_TO_UNICODE[7611] := 16#65F8;
   // GBK_TO_UNICODE[7612] := 16#9545;
   // GBK_TO_UNICODE[7613] := 16#65F9;
   // GBK_TO_UNICODE[7614] := 16#9546;
   // GBK_TO_UNICODE[7615] := 16#65FB;
   // GBK_TO_UNICODE[7616] := 16#9547;
   // GBK_TO_UNICODE[7617] := 16#65FC;
   // GBK_TO_UNICODE[7618] := 16#9548;
   // GBK_TO_UNICODE[7619] := 16#65FD;
   // GBK_TO_UNICODE[7620] := 16#9549;
   // GBK_TO_UNICODE[7621] := 16#65FE;
   // GBK_TO_UNICODE[7622] := 16#954A;
   // GBK_TO_UNICODE[7623] := 16#65FF;
   // GBK_TO_UNICODE[7624] := 16#954B;
   // GBK_TO_UNICODE[7625] := 16#6601;
   // GBK_TO_UNICODE[7626] := 16#954C;
   // GBK_TO_UNICODE[7627] := 16#6604;
   // GBK_TO_UNICODE[7628] := 16#954D;
   // GBK_TO_UNICODE[7629] := 16#6605;
   // GBK_TO_UNICODE[7630] := 16#954E;
   // GBK_TO_UNICODE[7631] := 16#6607;
   // GBK_TO_UNICODE[7632] := 16#954F;
   // GBK_TO_UNICODE[7633] := 16#6608;
   // GBK_TO_UNICODE[7634] := 16#9550;
   // GBK_TO_UNICODE[7635] := 16#6609;
   // GBK_TO_UNICODE[7636] := 16#9551;
   // GBK_TO_UNICODE[7637] := 16#660B;
   // GBK_TO_UNICODE[7638] := 16#9552;
   // GBK_TO_UNICODE[7639] := 16#660D;
   // GBK_TO_UNICODE[7640] := 16#9553;
   // GBK_TO_UNICODE[7641] := 16#6610;
   // GBK_TO_UNICODE[7642] := 16#9554;
   // GBK_TO_UNICODE[7643] := 16#6611;
   // GBK_TO_UNICODE[7644] := 16#9555;
   // GBK_TO_UNICODE[7645] := 16#6612;
   // GBK_TO_UNICODE[7646] := 16#9556;
   // GBK_TO_UNICODE[7647] := 16#6616;
   // GBK_TO_UNICODE[7648] := 16#9557;
   // GBK_TO_UNICODE[7649] := 16#6617;
   // GBK_TO_UNICODE[7650] := 16#9558;
   // GBK_TO_UNICODE[7651] := 16#6618;
   // GBK_TO_UNICODE[7652] := 16#9559;
   // GBK_TO_UNICODE[7653] := 16#661A;
   // GBK_TO_UNICODE[7654] := 16#955A;
   // GBK_TO_UNICODE[7655] := 16#661B;
   // GBK_TO_UNICODE[7656] := 16#955B;
   // GBK_TO_UNICODE[7657] := 16#661C;
   // GBK_TO_UNICODE[7658] := 16#955C;
   // GBK_TO_UNICODE[7659] := 16#661E;
   // GBK_TO_UNICODE[7660] := 16#955D;
   // GBK_TO_UNICODE[7661] := 16#6621;
   // GBK_TO_UNICODE[7662] := 16#955E;
   // GBK_TO_UNICODE[7663] := 16#6622;
   // GBK_TO_UNICODE[7664] := 16#955F;
   // GBK_TO_UNICODE[7665] := 16#6623;
   // GBK_TO_UNICODE[7666] := 16#9560;
   // GBK_TO_UNICODE[7667] := 16#6624;
   // GBK_TO_UNICODE[7668] := 16#9561;
   // GBK_TO_UNICODE[7669] := 16#6626;
   // GBK_TO_UNICODE[7670] := 16#9562;
   // GBK_TO_UNICODE[7671] := 16#6629;
   // GBK_TO_UNICODE[7672] := 16#9563;
   // GBK_TO_UNICODE[7673] := 16#662A;
   // GBK_TO_UNICODE[7674] := 16#9564;
   // GBK_TO_UNICODE[7675] := 16#662B;
   // GBK_TO_UNICODE[7676] := 16#9565;
   // GBK_TO_UNICODE[7677] := 16#662C;
   // GBK_TO_UNICODE[7678] := 16#9566;
   // GBK_TO_UNICODE[7679] := 16#662E;
   // GBK_TO_UNICODE[7680] := 16#9567;
   // GBK_TO_UNICODE[7681] := 16#6630;
   // GBK_TO_UNICODE[7682] := 16#9568;
   // GBK_TO_UNICODE[7683] := 16#6632;
   // GBK_TO_UNICODE[7684] := 16#9569;
   // GBK_TO_UNICODE[7685] := 16#6633;
   // GBK_TO_UNICODE[7686] := 16#956A;
   // GBK_TO_UNICODE[7687] := 16#6637;
   // GBK_TO_UNICODE[7688] := 16#956B;
   // GBK_TO_UNICODE[7689] := 16#6638;
   // GBK_TO_UNICODE[7690] := 16#956C;
   // GBK_TO_UNICODE[7691] := 16#6639;
   // GBK_TO_UNICODE[7692] := 16#956D;
   // GBK_TO_UNICODE[7693] := 16#663A;
   // GBK_TO_UNICODE[7694] := 16#956E;
   // GBK_TO_UNICODE[7695] := 16#663B;
   // GBK_TO_UNICODE[7696] := 16#956F;
   // GBK_TO_UNICODE[7697] := 16#663D;
   // GBK_TO_UNICODE[7698] := 16#9570;
   // GBK_TO_UNICODE[7699] := 16#663F;
   // GBK_TO_UNICODE[7700] := 16#9571;
   // GBK_TO_UNICODE[7701] := 16#6640;
   // GBK_TO_UNICODE[7702] := 16#9572;
   // GBK_TO_UNICODE[7703] := 16#6642;
   // GBK_TO_UNICODE[7704] := 16#9573;
   // GBK_TO_UNICODE[7705] := 16#6644;
   // GBK_TO_UNICODE[7706] := 16#9574;
   // GBK_TO_UNICODE[7707] := 16#6645;
   // GBK_TO_UNICODE[7708] := 16#9575;
   // GBK_TO_UNICODE[7709] := 16#6646;
   // GBK_TO_UNICODE[7710] := 16#9576;
   // GBK_TO_UNICODE[7711] := 16#6647;
   // GBK_TO_UNICODE[7712] := 16#9577;
   // GBK_TO_UNICODE[7713] := 16#6648;
   // GBK_TO_UNICODE[7714] := 16#9578;
   // GBK_TO_UNICODE[7715] := 16#6649;
   // GBK_TO_UNICODE[7716] := 16#9579;
   // GBK_TO_UNICODE[7717] := 16#664A;
   // GBK_TO_UNICODE[7718] := 16#957A;
   // GBK_TO_UNICODE[7719] := 16#664D;
   // GBK_TO_UNICODE[7720] := 16#957B;
   // GBK_TO_UNICODE[7721] := 16#664E;
   // GBK_TO_UNICODE[7722] := 16#957C;
   // GBK_TO_UNICODE[7723] := 16#6650;
   // GBK_TO_UNICODE[7724] := 16#957D;
   // GBK_TO_UNICODE[7725] := 16#6651;
   // GBK_TO_UNICODE[7726] := 16#957E;
   // GBK_TO_UNICODE[7727] := 16#6658;
   // GBK_TO_UNICODE[7728] := 16#9580;
   // GBK_TO_UNICODE[7729] := 16#6659;
   // GBK_TO_UNICODE[7730] := 16#9581;
   // GBK_TO_UNICODE[7731] := 16#665B;
   // GBK_TO_UNICODE[7732] := 16#9582;
   // GBK_TO_UNICODE[7733] := 16#665C;
   // GBK_TO_UNICODE[7734] := 16#9583;
   // GBK_TO_UNICODE[7735] := 16#665D;
   // GBK_TO_UNICODE[7736] := 16#9584;
   // GBK_TO_UNICODE[7737] := 16#665E;
   // GBK_TO_UNICODE[7738] := 16#9585;
   // GBK_TO_UNICODE[7739] := 16#6660;
   // GBK_TO_UNICODE[7740] := 16#9586;
   // GBK_TO_UNICODE[7741] := 16#6662;
   // GBK_TO_UNICODE[7742] := 16#9587;
   // GBK_TO_UNICODE[7743] := 16#6663;
   // GBK_TO_UNICODE[7744] := 16#9588;
   // GBK_TO_UNICODE[7745] := 16#6665;
   // GBK_TO_UNICODE[7746] := 16#9589;
   // GBK_TO_UNICODE[7747] := 16#6667;
   // GBK_TO_UNICODE[7748] := 16#958A;
   // GBK_TO_UNICODE[7749] := 16#6669;
   // GBK_TO_UNICODE[7750] := 16#958B;
   // GBK_TO_UNICODE[7751] := 16#666A;
   // GBK_TO_UNICODE[7752] := 16#958C;
   // GBK_TO_UNICODE[7753] := 16#666B;
   // GBK_TO_UNICODE[7754] := 16#958D;
   // GBK_TO_UNICODE[7755] := 16#666C;
   // GBK_TO_UNICODE[7756] := 16#958E;
   // GBK_TO_UNICODE[7757] := 16#666D;
   // GBK_TO_UNICODE[7758] := 16#958F;
   // GBK_TO_UNICODE[7759] := 16#6671;
   // GBK_TO_UNICODE[7760] := 16#9590;
   // GBK_TO_UNICODE[7761] := 16#6672;
   // GBK_TO_UNICODE[7762] := 16#9591;
   // GBK_TO_UNICODE[7763] := 16#6673;
   // GBK_TO_UNICODE[7764] := 16#9592;
   // GBK_TO_UNICODE[7765] := 16#6675;
   // GBK_TO_UNICODE[7766] := 16#9593;
   // GBK_TO_UNICODE[7767] := 16#6678;
   // GBK_TO_UNICODE[7768] := 16#9594;
   // GBK_TO_UNICODE[7769] := 16#6679;
   // GBK_TO_UNICODE[7770] := 16#9595;
   // GBK_TO_UNICODE[7771] := 16#667B;
   // GBK_TO_UNICODE[7772] := 16#9596;
   // GBK_TO_UNICODE[7773] := 16#667C;
   // GBK_TO_UNICODE[7774] := 16#9597;
   // GBK_TO_UNICODE[7775] := 16#667D;
   // GBK_TO_UNICODE[7776] := 16#9598;
   // GBK_TO_UNICODE[7777] := 16#667F;
   // GBK_TO_UNICODE[7778] := 16#9599;
   // GBK_TO_UNICODE[7779] := 16#6680;
   // GBK_TO_UNICODE[7780] := 16#959A;
   // GBK_TO_UNICODE[7781] := 16#6681;
   // GBK_TO_UNICODE[7782] := 16#959B;
   // GBK_TO_UNICODE[7783] := 16#6683;
   // GBK_TO_UNICODE[7784] := 16#959C;
   // GBK_TO_UNICODE[7785] := 16#6685;
   // GBK_TO_UNICODE[7786] := 16#959D;
   // GBK_TO_UNICODE[7787] := 16#6686;
   // GBK_TO_UNICODE[7788] := 16#959E;
   // GBK_TO_UNICODE[7789] := 16#6688;
   // GBK_TO_UNICODE[7790] := 16#959F;
   // GBK_TO_UNICODE[7791] := 16#6689;
   // GBK_TO_UNICODE[7792] := 16#95A0;
   // GBK_TO_UNICODE[7793] := 16#668A;
   // GBK_TO_UNICODE[7794] := 16#95A1;
   // GBK_TO_UNICODE[7795] := 16#668B;
   // GBK_TO_UNICODE[7796] := 16#95A2;
   // GBK_TO_UNICODE[7797] := 16#668D;
   // GBK_TO_UNICODE[7798] := 16#95A3;
   // GBK_TO_UNICODE[7799] := 16#668E;
   // GBK_TO_UNICODE[7800] := 16#95A4;
   // GBK_TO_UNICODE[7801] := 16#668F;
   // GBK_TO_UNICODE[7802] := 16#95A5;
   // GBK_TO_UNICODE[7803] := 16#6690;
   // GBK_TO_UNICODE[7804] := 16#95A6;
   // GBK_TO_UNICODE[7805] := 16#6692;
   // GBK_TO_UNICODE[7806] := 16#95A7;
   // GBK_TO_UNICODE[7807] := 16#6693;
   // GBK_TO_UNICODE[7808] := 16#95A8;
   // GBK_TO_UNICODE[7809] := 16#6694;
   // GBK_TO_UNICODE[7810] := 16#95A9;
   // GBK_TO_UNICODE[7811] := 16#6695;
   // GBK_TO_UNICODE[7812] := 16#95AA;
   // GBK_TO_UNICODE[7813] := 16#6698;
   // GBK_TO_UNICODE[7814] := 16#95AB;
   // GBK_TO_UNICODE[7815] := 16#6699;
   // GBK_TO_UNICODE[7816] := 16#95AC;
   // GBK_TO_UNICODE[7817] := 16#669A;
   // GBK_TO_UNICODE[7818] := 16#95AD;
   // GBK_TO_UNICODE[7819] := 16#669B;
   // GBK_TO_UNICODE[7820] := 16#95AE;
   // GBK_TO_UNICODE[7821] := 16#669C;
   // GBK_TO_UNICODE[7822] := 16#95AF;
   // GBK_TO_UNICODE[7823] := 16#669E;
   // GBK_TO_UNICODE[7824] := 16#95B0;
   // GBK_TO_UNICODE[7825] := 16#669F;
   // GBK_TO_UNICODE[7826] := 16#95B1;
   // GBK_TO_UNICODE[7827] := 16#66A0;
   // GBK_TO_UNICODE[7828] := 16#95B2;
   // GBK_TO_UNICODE[7829] := 16#66A1;
   // GBK_TO_UNICODE[7830] := 16#95B3;
   // GBK_TO_UNICODE[7831] := 16#66A2;
   // GBK_TO_UNICODE[7832] := 16#95B4;
   // GBK_TO_UNICODE[7833] := 16#66A3;
   // GBK_TO_UNICODE[7834] := 16#95B5;
   // GBK_TO_UNICODE[7835] := 16#66A4;
   // GBK_TO_UNICODE[7836] := 16#95B6;
   // GBK_TO_UNICODE[7837] := 16#66A5;
   // GBK_TO_UNICODE[7838] := 16#95B7;
   // GBK_TO_UNICODE[7839] := 16#66A6;
   // GBK_TO_UNICODE[7840] := 16#95B8;
   // GBK_TO_UNICODE[7841] := 16#66A9;
   // GBK_TO_UNICODE[7842] := 16#95B9;
   // GBK_TO_UNICODE[7843] := 16#66AA;
   // GBK_TO_UNICODE[7844] := 16#95BA;
   // GBK_TO_UNICODE[7845] := 16#66AB;
   // GBK_TO_UNICODE[7846] := 16#95BB;
   // GBK_TO_UNICODE[7847] := 16#66AC;
   // GBK_TO_UNICODE[7848] := 16#95BC;
   // GBK_TO_UNICODE[7849] := 16#66AD;
   // GBK_TO_UNICODE[7850] := 16#95BD;
   // GBK_TO_UNICODE[7851] := 16#66AF;
   // GBK_TO_UNICODE[7852] := 16#95BE;
   // GBK_TO_UNICODE[7853] := 16#66B0;
   // GBK_TO_UNICODE[7854] := 16#95BF;
   // GBK_TO_UNICODE[7855] := 16#66B1;
   // GBK_TO_UNICODE[7856] := 16#95C0;
   // GBK_TO_UNICODE[7857] := 16#66B2;
   // GBK_TO_UNICODE[7858] := 16#95C1;
   // GBK_TO_UNICODE[7859] := 16#66B3;
   // GBK_TO_UNICODE[7860] := 16#95C2;
   // GBK_TO_UNICODE[7861] := 16#66B5;
   // GBK_TO_UNICODE[7862] := 16#95C3;
   // GBK_TO_UNICODE[7863] := 16#66B6;
   // GBK_TO_UNICODE[7864] := 16#95C4;
   // GBK_TO_UNICODE[7865] := 16#66B7;
   // GBK_TO_UNICODE[7866] := 16#95C5;
   // GBK_TO_UNICODE[7867] := 16#66B8;
   // GBK_TO_UNICODE[7868] := 16#95C6;
   // GBK_TO_UNICODE[7869] := 16#66BA;
   // GBK_TO_UNICODE[7870] := 16#95C7;
   // GBK_TO_UNICODE[7871] := 16#66BB;
   // GBK_TO_UNICODE[7872] := 16#95C8;
   // GBK_TO_UNICODE[7873] := 16#66BC;
   // GBK_TO_UNICODE[7874] := 16#95C9;
   // GBK_TO_UNICODE[7875] := 16#66BD;
   // GBK_TO_UNICODE[7876] := 16#95CA;
   // GBK_TO_UNICODE[7877] := 16#66BF;
   // GBK_TO_UNICODE[7878] := 16#95CB;
   // GBK_TO_UNICODE[7879] := 16#66C0;
   // GBK_TO_UNICODE[7880] := 16#95CC;
   // GBK_TO_UNICODE[7881] := 16#66C1;
   // GBK_TO_UNICODE[7882] := 16#95CD;
   // GBK_TO_UNICODE[7883] := 16#66C2;
   // GBK_TO_UNICODE[7884] := 16#95CE;
   // GBK_TO_UNICODE[7885] := 16#66C3;
   // GBK_TO_UNICODE[7886] := 16#95CF;
   // GBK_TO_UNICODE[7887] := 16#66C4;
   // GBK_TO_UNICODE[7888] := 16#95D0;
   // GBK_TO_UNICODE[7889] := 16#66C5;
   // GBK_TO_UNICODE[7890] := 16#95D1;
   // GBK_TO_UNICODE[7891] := 16#66C6;
   // GBK_TO_UNICODE[7892] := 16#95D2;
   // GBK_TO_UNICODE[7893] := 16#66C7;
   // GBK_TO_UNICODE[7894] := 16#95D3;
   // GBK_TO_UNICODE[7895] := 16#66C8;
   // GBK_TO_UNICODE[7896] := 16#95D4;
   // GBK_TO_UNICODE[7897] := 16#66C9;
   // GBK_TO_UNICODE[7898] := 16#95D5;
   // GBK_TO_UNICODE[7899] := 16#66CA;
   // GBK_TO_UNICODE[7900] := 16#95D6;
   // GBK_TO_UNICODE[7901] := 16#66CB;
   // GBK_TO_UNICODE[7902] := 16#95D7;
   // GBK_TO_UNICODE[7903] := 16#66CC;
   // GBK_TO_UNICODE[7904] := 16#95D8;
   // GBK_TO_UNICODE[7905] := 16#66CD;
   // GBK_TO_UNICODE[7906] := 16#95D9;
   // GBK_TO_UNICODE[7907] := 16#66CE;
   // GBK_TO_UNICODE[7908] := 16#95DA;
   // GBK_TO_UNICODE[7909] := 16#66CF;
   // GBK_TO_UNICODE[7910] := 16#95DB;
   // GBK_TO_UNICODE[7911] := 16#66D0;
   // GBK_TO_UNICODE[7912] := 16#95DC;
   // GBK_TO_UNICODE[7913] := 16#66D1;
   // GBK_TO_UNICODE[7914] := 16#95DD;
   // GBK_TO_UNICODE[7915] := 16#66D2;
   // GBK_TO_UNICODE[7916] := 16#95DE;
   // GBK_TO_UNICODE[7917] := 16#66D3;
   // GBK_TO_UNICODE[7918] := 16#95DF;
   // GBK_TO_UNICODE[7919] := 16#66D4;
   // GBK_TO_UNICODE[7920] := 16#95E0;
   // GBK_TO_UNICODE[7921] := 16#66D5;
   // GBK_TO_UNICODE[7922] := 16#95E1;
   // GBK_TO_UNICODE[7923] := 16#66D6;
   // GBK_TO_UNICODE[7924] := 16#95E2;
   // GBK_TO_UNICODE[7925] := 16#66D7;
   // GBK_TO_UNICODE[7926] := 16#95E3;
   // GBK_TO_UNICODE[7927] := 16#66D8;
   // GBK_TO_UNICODE[7928] := 16#95E4;
   // GBK_TO_UNICODE[7929] := 16#66DA;
   // GBK_TO_UNICODE[7930] := 16#95E5;
   // GBK_TO_UNICODE[7931] := 16#66DE;
   // GBK_TO_UNICODE[7932] := 16#95E6;
   // GBK_TO_UNICODE[7933] := 16#66DF;
   // GBK_TO_UNICODE[7934] := 16#95E7;
   // GBK_TO_UNICODE[7935] := 16#66E0;
   // GBK_TO_UNICODE[7936] := 16#95E8;
   // GBK_TO_UNICODE[7937] := 16#66E1;
   // GBK_TO_UNICODE[7938] := 16#95E9;
   // GBK_TO_UNICODE[7939] := 16#66E2;
   // GBK_TO_UNICODE[7940] := 16#95EA;
   // GBK_TO_UNICODE[7941] := 16#66E3;
   // GBK_TO_UNICODE[7942] := 16#95EB;
   // GBK_TO_UNICODE[7943] := 16#66E4;
   // GBK_TO_UNICODE[7944] := 16#95EC;
   // GBK_TO_UNICODE[7945] := 16#66E5;
   // GBK_TO_UNICODE[7946] := 16#95ED;
   // GBK_TO_UNICODE[7947] := 16#66E7;
   // GBK_TO_UNICODE[7948] := 16#95EE;
   // GBK_TO_UNICODE[7949] := 16#66E8;
   // GBK_TO_UNICODE[7950] := 16#95EF;
   // GBK_TO_UNICODE[7951] := 16#66EA;
   // GBK_TO_UNICODE[7952] := 16#95F0;
   // GBK_TO_UNICODE[7953] := 16#66EB;
   // GBK_TO_UNICODE[7954] := 16#95F1;
   // GBK_TO_UNICODE[7955] := 16#66EC;
   // GBK_TO_UNICODE[7956] := 16#95F2;
   // GBK_TO_UNICODE[7957] := 16#66ED;
   // GBK_TO_UNICODE[7958] := 16#95F3;
   // GBK_TO_UNICODE[7959] := 16#66EE;
   // GBK_TO_UNICODE[7960] := 16#95F4;
   // GBK_TO_UNICODE[7961] := 16#66EF;
   // GBK_TO_UNICODE[7962] := 16#95F5;
   // GBK_TO_UNICODE[7963] := 16#66F1;
   // GBK_TO_UNICODE[7964] := 16#95F6;
   // GBK_TO_UNICODE[7965] := 16#66F5;
   // GBK_TO_UNICODE[7966] := 16#95F7;
   // GBK_TO_UNICODE[7967] := 16#66F6;
   // GBK_TO_UNICODE[7968] := 16#95F8;
   // GBK_TO_UNICODE[7969] := 16#66F8;
   // GBK_TO_UNICODE[7970] := 16#95F9;
   // GBK_TO_UNICODE[7971] := 16#66FA;
   // GBK_TO_UNICODE[7972] := 16#95FA;
   // GBK_TO_UNICODE[7973] := 16#66FB;
   // GBK_TO_UNICODE[7974] := 16#95FB;
   // GBK_TO_UNICODE[7975] := 16#66FD;
   // GBK_TO_UNICODE[7976] := 16#95FC;
   // GBK_TO_UNICODE[7977] := 16#6701;
   // GBK_TO_UNICODE[7978] := 16#95FD;
   // GBK_TO_UNICODE[7979] := 16#6702;
   // GBK_TO_UNICODE[7980] := 16#95FE;
   // GBK_TO_UNICODE[7981] := 16#6703;
   // GBK_TO_UNICODE[7982] := 16#9640;
   // GBK_TO_UNICODE[7983] := 16#6704;
   // GBK_TO_UNICODE[7984] := 16#9641;
   // GBK_TO_UNICODE[7985] := 16#6705;
   // GBK_TO_UNICODE[7986] := 16#9642;
   // GBK_TO_UNICODE[7987] := 16#6706;
   // GBK_TO_UNICODE[7988] := 16#9643;
   // GBK_TO_UNICODE[7989] := 16#6707;
   // GBK_TO_UNICODE[7990] := 16#9644;
   // GBK_TO_UNICODE[7991] := 16#670C;
   // GBK_TO_UNICODE[7992] := 16#9645;
   // GBK_TO_UNICODE[7993] := 16#670E;
   // GBK_TO_UNICODE[7994] := 16#9646;
   // GBK_TO_UNICODE[7995] := 16#670F;
   // GBK_TO_UNICODE[7996] := 16#9647;
   // GBK_TO_UNICODE[7997] := 16#6711;
   // GBK_TO_UNICODE[7998] := 16#9648;
   // GBK_TO_UNICODE[7999] := 16#6712;
   // GBK_TO_UNICODE[8000] := 16#9649;
   // GBK_TO_UNICODE[8001] := 16#6713;
   // GBK_TO_UNICODE[8002] := 16#964A;
   // GBK_TO_UNICODE[8003] := 16#6716;
   // GBK_TO_UNICODE[8004] := 16#964B;
   // GBK_TO_UNICODE[8005] := 16#6718;
   // GBK_TO_UNICODE[8006] := 16#964C;
   // GBK_TO_UNICODE[8007] := 16#6719;
   // GBK_TO_UNICODE[8008] := 16#964D;
   // GBK_TO_UNICODE[8009] := 16#671A;
   // GBK_TO_UNICODE[8010] := 16#964E;
   // GBK_TO_UNICODE[8011] := 16#671C;
   // GBK_TO_UNICODE[8012] := 16#964F;
   // GBK_TO_UNICODE[8013] := 16#671E;
   // GBK_TO_UNICODE[8014] := 16#9650;
   // GBK_TO_UNICODE[8015] := 16#6720;
   // GBK_TO_UNICODE[8016] := 16#9651;
   // GBK_TO_UNICODE[8017] := 16#6721;
   // GBK_TO_UNICODE[8018] := 16#9652;
   // GBK_TO_UNICODE[8019] := 16#6722;
   // GBK_TO_UNICODE[8020] := 16#9653;
   // GBK_TO_UNICODE[8021] := 16#6723;
   // GBK_TO_UNICODE[8022] := 16#9654;
   // GBK_TO_UNICODE[8023] := 16#6724;
   // GBK_TO_UNICODE[8024] := 16#9655;
   // GBK_TO_UNICODE[8025] := 16#6725;
   // GBK_TO_UNICODE[8026] := 16#9656;
   // GBK_TO_UNICODE[8027] := 16#6727;
   // GBK_TO_UNICODE[8028] := 16#9657;
   // GBK_TO_UNICODE[8029] := 16#6729;
   // GBK_TO_UNICODE[8030] := 16#9658;
   // GBK_TO_UNICODE[8031] := 16#672E;
   // GBK_TO_UNICODE[8032] := 16#9659;
   // GBK_TO_UNICODE[8033] := 16#6730;
   // GBK_TO_UNICODE[8034] := 16#965A;
   // GBK_TO_UNICODE[8035] := 16#6732;
   // GBK_TO_UNICODE[8036] := 16#965B;
   // GBK_TO_UNICODE[8037] := 16#6733;
   // GBK_TO_UNICODE[8038] := 16#965C;
   // GBK_TO_UNICODE[8039] := 16#6736;
   // GBK_TO_UNICODE[8040] := 16#965D;
   // GBK_TO_UNICODE[8041] := 16#6737;
   // GBK_TO_UNICODE[8042] := 16#965E;
   // GBK_TO_UNICODE[8043] := 16#6738;
   // GBK_TO_UNICODE[8044] := 16#965F;
   // GBK_TO_UNICODE[8045] := 16#6739;
   // GBK_TO_UNICODE[8046] := 16#9660;
   // GBK_TO_UNICODE[8047] := 16#673B;
   // GBK_TO_UNICODE[8048] := 16#9661;
   // GBK_TO_UNICODE[8049] := 16#673C;
   // GBK_TO_UNICODE[8050] := 16#9662;
   // GBK_TO_UNICODE[8051] := 16#673E;
   // GBK_TO_UNICODE[8052] := 16#9663;
   // GBK_TO_UNICODE[8053] := 16#673F;
   // GBK_TO_UNICODE[8054] := 16#9664;
   // GBK_TO_UNICODE[8055] := 16#6741;
   // GBK_TO_UNICODE[8056] := 16#9665;
   // GBK_TO_UNICODE[8057] := 16#6744;
   // GBK_TO_UNICODE[8058] := 16#9666;
   // GBK_TO_UNICODE[8059] := 16#6745;
   // GBK_TO_UNICODE[8060] := 16#9667;
   // GBK_TO_UNICODE[8061] := 16#6747;
   // GBK_TO_UNICODE[8062] := 16#9668;
   // GBK_TO_UNICODE[8063] := 16#674A;
   // GBK_TO_UNICODE[8064] := 16#9669;
   // GBK_TO_UNICODE[8065] := 16#674B;
   // GBK_TO_UNICODE[8066] := 16#966A;
   // GBK_TO_UNICODE[8067] := 16#674D;
   // GBK_TO_UNICODE[8068] := 16#966B;
   // GBK_TO_UNICODE[8069] := 16#6752;
   // GBK_TO_UNICODE[8070] := 16#966C;
   // GBK_TO_UNICODE[8071] := 16#6754;
   // GBK_TO_UNICODE[8072] := 16#966D;
   // GBK_TO_UNICODE[8073] := 16#6755;
   // GBK_TO_UNICODE[8074] := 16#966E;
   // GBK_TO_UNICODE[8075] := 16#6757;
   // GBK_TO_UNICODE[8076] := 16#966F;
   // GBK_TO_UNICODE[8077] := 16#6758;
   // GBK_TO_UNICODE[8078] := 16#9670;
   // GBK_TO_UNICODE[8079] := 16#6759;
   // GBK_TO_UNICODE[8080] := 16#9671;
   // GBK_TO_UNICODE[8081] := 16#675A;
   // GBK_TO_UNICODE[8082] := 16#9672;
   // GBK_TO_UNICODE[8083] := 16#675B;
   // GBK_TO_UNICODE[8084] := 16#9673;
   // GBK_TO_UNICODE[8085] := 16#675D;
   // GBK_TO_UNICODE[8086] := 16#9674;
   // GBK_TO_UNICODE[8087] := 16#6762;
   // GBK_TO_UNICODE[8088] := 16#9675;
   // GBK_TO_UNICODE[8089] := 16#6763;
   // GBK_TO_UNICODE[8090] := 16#9676;
   // GBK_TO_UNICODE[8091] := 16#6764;
   // GBK_TO_UNICODE[8092] := 16#9677;
   // GBK_TO_UNICODE[8093] := 16#6766;
   // GBK_TO_UNICODE[8094] := 16#9678;
   // GBK_TO_UNICODE[8095] := 16#6767;
   // GBK_TO_UNICODE[8096] := 16#9679;
   // GBK_TO_UNICODE[8097] := 16#676B;
   // GBK_TO_UNICODE[8098] := 16#967A;
   // GBK_TO_UNICODE[8099] := 16#676C;
   // GBK_TO_UNICODE[8100] := 16#967B;
   // GBK_TO_UNICODE[8101] := 16#676E;
   // GBK_TO_UNICODE[8102] := 16#967C;
   // GBK_TO_UNICODE[8103] := 16#6771;
   // GBK_TO_UNICODE[8104] := 16#967D;
   // GBK_TO_UNICODE[8105] := 16#6774;
   // GBK_TO_UNICODE[8106] := 16#967E;
   // GBK_TO_UNICODE[8107] := 16#6776;
   // GBK_TO_UNICODE[8108] := 16#9680;
   // GBK_TO_UNICODE[8109] := 16#6778;
   // GBK_TO_UNICODE[8110] := 16#9681;
   // GBK_TO_UNICODE[8111] := 16#6779;
   // GBK_TO_UNICODE[8112] := 16#9682;
   // GBK_TO_UNICODE[8113] := 16#677A;
   // GBK_TO_UNICODE[8114] := 16#9683;
   // GBK_TO_UNICODE[8115] := 16#677B;
   // GBK_TO_UNICODE[8116] := 16#9684;
   // GBK_TO_UNICODE[8117] := 16#677D;
   // GBK_TO_UNICODE[8118] := 16#9685;
   // GBK_TO_UNICODE[8119] := 16#6780;
   // GBK_TO_UNICODE[8120] := 16#9686;
   // GBK_TO_UNICODE[8121] := 16#6782;
   // GBK_TO_UNICODE[8122] := 16#9687;
   // GBK_TO_UNICODE[8123] := 16#6783;
   // GBK_TO_UNICODE[8124] := 16#9688;
   // GBK_TO_UNICODE[8125] := 16#6785;
   // GBK_TO_UNICODE[8126] := 16#9689;
   // GBK_TO_UNICODE[8127] := 16#6786;
   // GBK_TO_UNICODE[8128] := 16#968A;
   // GBK_TO_UNICODE[8129] := 16#6788;
   // GBK_TO_UNICODE[8130] := 16#968B;
   // GBK_TO_UNICODE[8131] := 16#678A;
   // GBK_TO_UNICODE[8132] := 16#968C;
   // GBK_TO_UNICODE[8133] := 16#678C;
   // GBK_TO_UNICODE[8134] := 16#968D;
   // GBK_TO_UNICODE[8135] := 16#678D;
   // GBK_TO_UNICODE[8136] := 16#968E;
   // GBK_TO_UNICODE[8137] := 16#678E;
   // GBK_TO_UNICODE[8138] := 16#968F;
   // GBK_TO_UNICODE[8139] := 16#678F;
   // GBK_TO_UNICODE[8140] := 16#9690;
   // GBK_TO_UNICODE[8141] := 16#6791;
   // GBK_TO_UNICODE[8142] := 16#9691;
   // GBK_TO_UNICODE[8143] := 16#6792;
   // GBK_TO_UNICODE[8144] := 16#9692;
   // GBK_TO_UNICODE[8145] := 16#6793;
   // GBK_TO_UNICODE[8146] := 16#9693;
   // GBK_TO_UNICODE[8147] := 16#6794;
   // GBK_TO_UNICODE[8148] := 16#9694;
   // GBK_TO_UNICODE[8149] := 16#6796;
   // GBK_TO_UNICODE[8150] := 16#9695;
   // GBK_TO_UNICODE[8151] := 16#6799;
   // GBK_TO_UNICODE[8152] := 16#9696;
   // GBK_TO_UNICODE[8153] := 16#679B;
   // GBK_TO_UNICODE[8154] := 16#9697;
   // GBK_TO_UNICODE[8155] := 16#679F;
   // GBK_TO_UNICODE[8156] := 16#9698;
   // GBK_TO_UNICODE[8157] := 16#67A0;
   // GBK_TO_UNICODE[8158] := 16#9699;
   // GBK_TO_UNICODE[8159] := 16#67A1;
   // GBK_TO_UNICODE[8160] := 16#969A;
   // GBK_TO_UNICODE[8161] := 16#67A4;
   // GBK_TO_UNICODE[8162] := 16#969B;
   // GBK_TO_UNICODE[8163] := 16#67A6;
   // GBK_TO_UNICODE[8164] := 16#969C;
   // GBK_TO_UNICODE[8165] := 16#67A9;
   // GBK_TO_UNICODE[8166] := 16#969D;
   // GBK_TO_UNICODE[8167] := 16#67AC;
   // GBK_TO_UNICODE[8168] := 16#969E;
   // GBK_TO_UNICODE[8169] := 16#67AE;
   // GBK_TO_UNICODE[8170] := 16#969F;
   // GBK_TO_UNICODE[8171] := 16#67B1;
   // GBK_TO_UNICODE[8172] := 16#96A0;
   // GBK_TO_UNICODE[8173] := 16#67B2;
   // GBK_TO_UNICODE[8174] := 16#96A1;
   // GBK_TO_UNICODE[8175] := 16#67B4;
   // GBK_TO_UNICODE[8176] := 16#96A2;
   // GBK_TO_UNICODE[8177] := 16#67B9;
   // GBK_TO_UNICODE[8178] := 16#96A3;
   // GBK_TO_UNICODE[8179] := 16#67BA;
   // GBK_TO_UNICODE[8180] := 16#96A4;
   // GBK_TO_UNICODE[8181] := 16#67BB;
   // GBK_TO_UNICODE[8182] := 16#96A5;
   // GBK_TO_UNICODE[8183] := 16#67BC;
   // GBK_TO_UNICODE[8184] := 16#96A6;
   // GBK_TO_UNICODE[8185] := 16#67BD;
   // GBK_TO_UNICODE[8186] := 16#96A7;
   // GBK_TO_UNICODE[8187] := 16#67BE;
   // GBK_TO_UNICODE[8188] := 16#96A8;
   // GBK_TO_UNICODE[8189] := 16#67BF;
   // GBK_TO_UNICODE[8190] := 16#96A9;
   // GBK_TO_UNICODE[8191] := 16#67C0;
   // GBK_TO_UNICODE[8192] := 16#96AA;
   // GBK_TO_UNICODE[8193] := 16#67C2;
   // GBK_TO_UNICODE[8194] := 16#96AB;
   // GBK_TO_UNICODE[8195] := 16#67C5;
   // GBK_TO_UNICODE[8196] := 16#96AC;
   // GBK_TO_UNICODE[8197] := 16#67C6;
   // GBK_TO_UNICODE[8198] := 16#96AD;
   // GBK_TO_UNICODE[8199] := 16#67C7;
   // GBK_TO_UNICODE[8200] := 16#96AE;
   // GBK_TO_UNICODE[8201] := 16#67C8;
   // GBK_TO_UNICODE[8202] := 16#96AF;
   // GBK_TO_UNICODE[8203] := 16#67C9;
   // GBK_TO_UNICODE[8204] := 16#96B0;
   // GBK_TO_UNICODE[8205] := 16#67CA;
   // GBK_TO_UNICODE[8206] := 16#96B1;
   // GBK_TO_UNICODE[8207] := 16#67CB;
   // GBK_TO_UNICODE[8208] := 16#96B2;
   // GBK_TO_UNICODE[8209] := 16#67CC;
   // GBK_TO_UNICODE[8210] := 16#96B3;
   // GBK_TO_UNICODE[8211] := 16#67CD;
   // GBK_TO_UNICODE[8212] := 16#96B4;
   // GBK_TO_UNICODE[8213] := 16#67CE;
   // GBK_TO_UNICODE[8214] := 16#96B5;
   // GBK_TO_UNICODE[8215] := 16#67D5;
   // GBK_TO_UNICODE[8216] := 16#96B6;
   // GBK_TO_UNICODE[8217] := 16#67D6;
   // GBK_TO_UNICODE[8218] := 16#96B7;
   // GBK_TO_UNICODE[8219] := 16#67D7;
   // GBK_TO_UNICODE[8220] := 16#96B8;
   // GBK_TO_UNICODE[8221] := 16#67DB;
   // GBK_TO_UNICODE[8222] := 16#96B9;
   // GBK_TO_UNICODE[8223] := 16#67DF;
   // GBK_TO_UNICODE[8224] := 16#96BA;
   // GBK_TO_UNICODE[8225] := 16#67E1;
   // GBK_TO_UNICODE[8226] := 16#96BB;
   // GBK_TO_UNICODE[8227] := 16#67E3;
   // GBK_TO_UNICODE[8228] := 16#96BC;
   // GBK_TO_UNICODE[8229] := 16#67E4;
   // GBK_TO_UNICODE[8230] := 16#96BD;
   // GBK_TO_UNICODE[8231] := 16#67E6;
   // GBK_TO_UNICODE[8232] := 16#96BE;
   // GBK_TO_UNICODE[8233] := 16#67E7;
   // GBK_TO_UNICODE[8234] := 16#96BF;
   // GBK_TO_UNICODE[8235] := 16#67E8;
   // GBK_TO_UNICODE[8236] := 16#96C0;
   // GBK_TO_UNICODE[8237] := 16#67EA;
   // GBK_TO_UNICODE[8238] := 16#96C1;
   // GBK_TO_UNICODE[8239] := 16#67EB;
   // GBK_TO_UNICODE[8240] := 16#96C2;
   // GBK_TO_UNICODE[8241] := 16#67ED;
   // GBK_TO_UNICODE[8242] := 16#96C3;
   // GBK_TO_UNICODE[8243] := 16#67EE;
   // GBK_TO_UNICODE[8244] := 16#96C4;
   // GBK_TO_UNICODE[8245] := 16#67F2;
   // GBK_TO_UNICODE[8246] := 16#96C5;
   // GBK_TO_UNICODE[8247] := 16#67F5;
   // GBK_TO_UNICODE[8248] := 16#96C6;
   // GBK_TO_UNICODE[8249] := 16#67F6;
   // GBK_TO_UNICODE[8250] := 16#96C7;
   // GBK_TO_UNICODE[8251] := 16#67F7;
   // GBK_TO_UNICODE[8252] := 16#96C8;
   // GBK_TO_UNICODE[8253] := 16#67F8;
   // GBK_TO_UNICODE[8254] := 16#96C9;
   // GBK_TO_UNICODE[8255] := 16#67F9;
   // GBK_TO_UNICODE[8256] := 16#96CA;
   // GBK_TO_UNICODE[8257] := 16#67FA;
   // GBK_TO_UNICODE[8258] := 16#96CB;
   // GBK_TO_UNICODE[8259] := 16#67FB;
   // GBK_TO_UNICODE[8260] := 16#96CC;
   // GBK_TO_UNICODE[8261] := 16#67FC;
   // GBK_TO_UNICODE[8262] := 16#96CD;
   // GBK_TO_UNICODE[8263] := 16#67FE;
   // GBK_TO_UNICODE[8264] := 16#96CE;
   // GBK_TO_UNICODE[8265] := 16#6801;
   // GBK_TO_UNICODE[8266] := 16#96CF;
   // GBK_TO_UNICODE[8267] := 16#6802;
   // GBK_TO_UNICODE[8268] := 16#96D0;
   // GBK_TO_UNICODE[8269] := 16#6803;
   // GBK_TO_UNICODE[8270] := 16#96D1;
   // GBK_TO_UNICODE[8271] := 16#6804;
   // GBK_TO_UNICODE[8272] := 16#96D2;
   // GBK_TO_UNICODE[8273] := 16#6806;
   // GBK_TO_UNICODE[8274] := 16#96D3;
   // GBK_TO_UNICODE[8275] := 16#680D;
   // GBK_TO_UNICODE[8276] := 16#96D4;
   // GBK_TO_UNICODE[8277] := 16#6810;
   // GBK_TO_UNICODE[8278] := 16#96D5;
   // GBK_TO_UNICODE[8279] := 16#6812;
   // GBK_TO_UNICODE[8280] := 16#96D6;
   // GBK_TO_UNICODE[8281] := 16#6814;
   // GBK_TO_UNICODE[8282] := 16#96D7;
   // GBK_TO_UNICODE[8283] := 16#6815;
   // GBK_TO_UNICODE[8284] := 16#96D8;
   // GBK_TO_UNICODE[8285] := 16#6818;
   // GBK_TO_UNICODE[8286] := 16#96D9;
   // GBK_TO_UNICODE[8287] := 16#6819;
   // GBK_TO_UNICODE[8288] := 16#96DA;
   // GBK_TO_UNICODE[8289] := 16#681A;
   // GBK_TO_UNICODE[8290] := 16#96DB;
   // GBK_TO_UNICODE[8291] := 16#681B;
   // GBK_TO_UNICODE[8292] := 16#96DC;
   // GBK_TO_UNICODE[8293] := 16#681C;
   // GBK_TO_UNICODE[8294] := 16#96DD;
   // GBK_TO_UNICODE[8295] := 16#681E;
   // GBK_TO_UNICODE[8296] := 16#96DE;
   // GBK_TO_UNICODE[8297] := 16#681F;
   // GBK_TO_UNICODE[8298] := 16#96DF;
   // GBK_TO_UNICODE[8299] := 16#6820;
   // GBK_TO_UNICODE[8300] := 16#96E0;
   // GBK_TO_UNICODE[8301] := 16#6822;
   // GBK_TO_UNICODE[8302] := 16#96E1;
   // GBK_TO_UNICODE[8303] := 16#6823;
   // GBK_TO_UNICODE[8304] := 16#96E2;
   // GBK_TO_UNICODE[8305] := 16#6824;
   // GBK_TO_UNICODE[8306] := 16#96E3;
   // GBK_TO_UNICODE[8307] := 16#6825;
   // GBK_TO_UNICODE[8308] := 16#96E4;
   // GBK_TO_UNICODE[8309] := 16#6826;
   // GBK_TO_UNICODE[8310] := 16#96E5;
   // GBK_TO_UNICODE[8311] := 16#6827;
   // GBK_TO_UNICODE[8312] := 16#96E6;
   // GBK_TO_UNICODE[8313] := 16#6828;
   // GBK_TO_UNICODE[8314] := 16#96E7;
   // GBK_TO_UNICODE[8315] := 16#682B;
   // GBK_TO_UNICODE[8316] := 16#96E8;
   // GBK_TO_UNICODE[8317] := 16#682C;
   // GBK_TO_UNICODE[8318] := 16#96E9;
   // GBK_TO_UNICODE[8319] := 16#682D;
   // GBK_TO_UNICODE[8320] := 16#96EA;
   // GBK_TO_UNICODE[8321] := 16#682E;
   // GBK_TO_UNICODE[8322] := 16#96EB;
   // GBK_TO_UNICODE[8323] := 16#682F;
   // GBK_TO_UNICODE[8324] := 16#96EC;
   // GBK_TO_UNICODE[8325] := 16#6830;
   // GBK_TO_UNICODE[8326] := 16#96ED;
   // GBK_TO_UNICODE[8327] := 16#6831;
   // GBK_TO_UNICODE[8328] := 16#96EE;
   // GBK_TO_UNICODE[8329] := 16#6834;
   // GBK_TO_UNICODE[8330] := 16#96EF;
   // GBK_TO_UNICODE[8331] := 16#6835;
   // GBK_TO_UNICODE[8332] := 16#96F0;
   // GBK_TO_UNICODE[8333] := 16#6836;
   // GBK_TO_UNICODE[8334] := 16#96F1;
   // GBK_TO_UNICODE[8335] := 16#683A;
   // GBK_TO_UNICODE[8336] := 16#96F2;
   // GBK_TO_UNICODE[8337] := 16#683B;
   // GBK_TO_UNICODE[8338] := 16#96F3;
   // GBK_TO_UNICODE[8339] := 16#683F;
   // GBK_TO_UNICODE[8340] := 16#96F4;
   // GBK_TO_UNICODE[8341] := 16#6847;
   // GBK_TO_UNICODE[8342] := 16#96F5;
   // GBK_TO_UNICODE[8343] := 16#684B;
   // GBK_TO_UNICODE[8344] := 16#96F6;
   // GBK_TO_UNICODE[8345] := 16#684D;
   // GBK_TO_UNICODE[8346] := 16#96F7;
   // GBK_TO_UNICODE[8347] := 16#684F;
   // GBK_TO_UNICODE[8348] := 16#96F8;
   // GBK_TO_UNICODE[8349] := 16#6852;
   // GBK_TO_UNICODE[8350] := 16#96F9;
   // GBK_TO_UNICODE[8351] := 16#6856;
   // GBK_TO_UNICODE[8352] := 16#96FA;
   // GBK_TO_UNICODE[8353] := 16#6857;
   // GBK_TO_UNICODE[8354] := 16#96FB;
   // GBK_TO_UNICODE[8355] := 16#6858;
   // GBK_TO_UNICODE[8356] := 16#96FC;
   // GBK_TO_UNICODE[8357] := 16#6859;
   // GBK_TO_UNICODE[8358] := 16#96FD;
   // GBK_TO_UNICODE[8359] := 16#685A;
   // GBK_TO_UNICODE[8360] := 16#96FE;
   // GBK_TO_UNICODE[8361] := 16#685B;
   // GBK_TO_UNICODE[8362] := 16#9740;
   // GBK_TO_UNICODE[8363] := 16#685C;
   // GBK_TO_UNICODE[8364] := 16#9741;
   // GBK_TO_UNICODE[8365] := 16#685D;
   // GBK_TO_UNICODE[8366] := 16#9742;
   // GBK_TO_UNICODE[8367] := 16#685E;
   // GBK_TO_UNICODE[8368] := 16#9743;
   // GBK_TO_UNICODE[8369] := 16#685F;
   // GBK_TO_UNICODE[8370] := 16#9744;
   // GBK_TO_UNICODE[8371] := 16#686A;
   // GBK_TO_UNICODE[8372] := 16#9745;
   // GBK_TO_UNICODE[8373] := 16#686C;
   // GBK_TO_UNICODE[8374] := 16#9746;
   // GBK_TO_UNICODE[8375] := 16#686D;
   // GBK_TO_UNICODE[8376] := 16#9747;
   // GBK_TO_UNICODE[8377] := 16#686E;
   // GBK_TO_UNICODE[8378] := 16#9748;
   // GBK_TO_UNICODE[8379] := 16#686F;
   // GBK_TO_UNICODE[8380] := 16#9749;
   // GBK_TO_UNICODE[8381] := 16#6870;
   // GBK_TO_UNICODE[8382] := 16#974A;
   // GBK_TO_UNICODE[8383] := 16#6871;
   // GBK_TO_UNICODE[8384] := 16#974B;
   // GBK_TO_UNICODE[8385] := 16#6872;
   // GBK_TO_UNICODE[8386] := 16#974C;
   // GBK_TO_UNICODE[8387] := 16#6873;
   // GBK_TO_UNICODE[8388] := 16#974D;
   // GBK_TO_UNICODE[8389] := 16#6875;
   // GBK_TO_UNICODE[8390] := 16#974E;
   // GBK_TO_UNICODE[8391] := 16#6878;
   // GBK_TO_UNICODE[8392] := 16#974F;
   // GBK_TO_UNICODE[8393] := 16#6879;
   // GBK_TO_UNICODE[8394] := 16#9750;
   // GBK_TO_UNICODE[8395] := 16#687A;
   // GBK_TO_UNICODE[8396] := 16#9751;
   // GBK_TO_UNICODE[8397] := 16#687B;
   // GBK_TO_UNICODE[8398] := 16#9752;
   // GBK_TO_UNICODE[8399] := 16#687C;
   // GBK_TO_UNICODE[8400] := 16#9753;
   // GBK_TO_UNICODE[8401] := 16#687D;
   // GBK_TO_UNICODE[8402] := 16#9754;
   // GBK_TO_UNICODE[8403] := 16#687E;
   // GBK_TO_UNICODE[8404] := 16#9755;
   // GBK_TO_UNICODE[8405] := 16#687F;
   // GBK_TO_UNICODE[8406] := 16#9756;
   // GBK_TO_UNICODE[8407] := 16#6880;
   // GBK_TO_UNICODE[8408] := 16#9757;
   // GBK_TO_UNICODE[8409] := 16#6882;
   // GBK_TO_UNICODE[8410] := 16#9758;
   // GBK_TO_UNICODE[8411] := 16#6884;
   // GBK_TO_UNICODE[8412] := 16#9759;
   // GBK_TO_UNICODE[8413] := 16#6887;
   // GBK_TO_UNICODE[8414] := 16#975A;
   // GBK_TO_UNICODE[8415] := 16#6888;
   // GBK_TO_UNICODE[8416] := 16#975B;
   // GBK_TO_UNICODE[8417] := 16#6889;
   // GBK_TO_UNICODE[8418] := 16#975C;
   // GBK_TO_UNICODE[8419] := 16#688A;
   // GBK_TO_UNICODE[8420] := 16#975D;
   // GBK_TO_UNICODE[8421] := 16#688B;
   // GBK_TO_UNICODE[8422] := 16#975E;
   // GBK_TO_UNICODE[8423] := 16#688C;
   // GBK_TO_UNICODE[8424] := 16#975F;
   // GBK_TO_UNICODE[8425] := 16#688D;
   // GBK_TO_UNICODE[8426] := 16#9760;
   // GBK_TO_UNICODE[8427] := 16#688E;
   // GBK_TO_UNICODE[8428] := 16#9761;
   // GBK_TO_UNICODE[8429] := 16#6890;
   // GBK_TO_UNICODE[8430] := 16#9762;
   // GBK_TO_UNICODE[8431] := 16#6891;
   // GBK_TO_UNICODE[8432] := 16#9763;
   // GBK_TO_UNICODE[8433] := 16#6892;
   // GBK_TO_UNICODE[8434] := 16#9764;
   // GBK_TO_UNICODE[8435] := 16#6894;
   // GBK_TO_UNICODE[8436] := 16#9765;
   // GBK_TO_UNICODE[8437] := 16#6895;
   // GBK_TO_UNICODE[8438] := 16#9766;
   // GBK_TO_UNICODE[8439] := 16#6896;
   // GBK_TO_UNICODE[8440] := 16#9767;
   // GBK_TO_UNICODE[8441] := 16#6898;
   // GBK_TO_UNICODE[8442] := 16#9768;
   // GBK_TO_UNICODE[8443] := 16#6899;
   // GBK_TO_UNICODE[8444] := 16#9769;
   // GBK_TO_UNICODE[8445] := 16#689A;
   // GBK_TO_UNICODE[8446] := 16#976A;
   // GBK_TO_UNICODE[8447] := 16#689B;
   // GBK_TO_UNICODE[8448] := 16#976B;
   // GBK_TO_UNICODE[8449] := 16#689C;
   // GBK_TO_UNICODE[8450] := 16#976C;
   // GBK_TO_UNICODE[8451] := 16#689D;
   // GBK_TO_UNICODE[8452] := 16#976D;
   // GBK_TO_UNICODE[8453] := 16#689E;
   // GBK_TO_UNICODE[8454] := 16#976E;
   // GBK_TO_UNICODE[8455] := 16#689F;
   // GBK_TO_UNICODE[8456] := 16#976F;
   // GBK_TO_UNICODE[8457] := 16#68A0;
   // GBK_TO_UNICODE[8458] := 16#9770;
   // GBK_TO_UNICODE[8459] := 16#68A1;
   // GBK_TO_UNICODE[8460] := 16#9771;
   // GBK_TO_UNICODE[8461] := 16#68A3;
   // GBK_TO_UNICODE[8462] := 16#9772;
   // GBK_TO_UNICODE[8463] := 16#68A4;
   // GBK_TO_UNICODE[8464] := 16#9773;
   // GBK_TO_UNICODE[8465] := 16#68A5;
   // GBK_TO_UNICODE[8466] := 16#9774;
   // GBK_TO_UNICODE[8467] := 16#68A9;
   // GBK_TO_UNICODE[8468] := 16#9775;
   // GBK_TO_UNICODE[8469] := 16#68AA;
   // GBK_TO_UNICODE[8470] := 16#9776;
   // GBK_TO_UNICODE[8471] := 16#68AB;
   // GBK_TO_UNICODE[8472] := 16#9777;
   // GBK_TO_UNICODE[8473] := 16#68AC;
   // GBK_TO_UNICODE[8474] := 16#9778;
   // GBK_TO_UNICODE[8475] := 16#68AE;
   // GBK_TO_UNICODE[8476] := 16#9779;
   // GBK_TO_UNICODE[8477] := 16#68B1;
   // GBK_TO_UNICODE[8478] := 16#977A;
   // GBK_TO_UNICODE[8479] := 16#68B2;
   // GBK_TO_UNICODE[8480] := 16#977B;
   // GBK_TO_UNICODE[8481] := 16#68B4;
   // GBK_TO_UNICODE[8482] := 16#977C;
   // GBK_TO_UNICODE[8483] := 16#68B6;
   // GBK_TO_UNICODE[8484] := 16#977D;
   // GBK_TO_UNICODE[8485] := 16#68B7;
   // GBK_TO_UNICODE[8486] := 16#977E;
   // GBK_TO_UNICODE[8487] := 16#68B8;
   // GBK_TO_UNICODE[8488] := 16#9780;
   // GBK_TO_UNICODE[8489] := 16#68B9;
   // GBK_TO_UNICODE[8490] := 16#9781;
   // GBK_TO_UNICODE[8491] := 16#68BA;
   // GBK_TO_UNICODE[8492] := 16#9782;
   // GBK_TO_UNICODE[8493] := 16#68BB;
   // GBK_TO_UNICODE[8494] := 16#9783;
   // GBK_TO_UNICODE[8495] := 16#68BC;
   // GBK_TO_UNICODE[8496] := 16#9784;
   // GBK_TO_UNICODE[8497] := 16#68BD;
   // GBK_TO_UNICODE[8498] := 16#9785;
   // GBK_TO_UNICODE[8499] := 16#68BE;
   // GBK_TO_UNICODE[8500] := 16#9786;
   // GBK_TO_UNICODE[8501] := 16#68BF;
   // GBK_TO_UNICODE[8502] := 16#9787;
   // GBK_TO_UNICODE[8503] := 16#68C1;
   // GBK_TO_UNICODE[8504] := 16#9788;
   // GBK_TO_UNICODE[8505] := 16#68C3;
   // GBK_TO_UNICODE[8506] := 16#9789;
   // GBK_TO_UNICODE[8507] := 16#68C4;
   // GBK_TO_UNICODE[8508] := 16#978A;
   // GBK_TO_UNICODE[8509] := 16#68C5;
   // GBK_TO_UNICODE[8510] := 16#978B;
   // GBK_TO_UNICODE[8511] := 16#68C6;
   // GBK_TO_UNICODE[8512] := 16#978C;
   // GBK_TO_UNICODE[8513] := 16#68C7;
   // GBK_TO_UNICODE[8514] := 16#978D;
   // GBK_TO_UNICODE[8515] := 16#68C8;
   // GBK_TO_UNICODE[8516] := 16#978E;
   // GBK_TO_UNICODE[8517] := 16#68CA;
   // GBK_TO_UNICODE[8518] := 16#978F;
   // GBK_TO_UNICODE[8519] := 16#68CC;
   // GBK_TO_UNICODE[8520] := 16#9790;
   // GBK_TO_UNICODE[8521] := 16#68CE;
   // GBK_TO_UNICODE[8522] := 16#9791;
   // GBK_TO_UNICODE[8523] := 16#68CF;
   // GBK_TO_UNICODE[8524] := 16#9792;
   // GBK_TO_UNICODE[8525] := 16#68D0;
   // GBK_TO_UNICODE[8526] := 16#9793;
   // GBK_TO_UNICODE[8527] := 16#68D1;
   // GBK_TO_UNICODE[8528] := 16#9794;
   // GBK_TO_UNICODE[8529] := 16#68D3;
   // GBK_TO_UNICODE[8530] := 16#9795;
   // GBK_TO_UNICODE[8531] := 16#68D4;
   // GBK_TO_UNICODE[8532] := 16#9796;
   // GBK_TO_UNICODE[8533] := 16#68D6;
   // GBK_TO_UNICODE[8534] := 16#9797;
   // GBK_TO_UNICODE[8535] := 16#68D7;
   // GBK_TO_UNICODE[8536] := 16#9798;
   // GBK_TO_UNICODE[8537] := 16#68D9;
   // GBK_TO_UNICODE[8538] := 16#9799;
   // GBK_TO_UNICODE[8539] := 16#68DB;
   // GBK_TO_UNICODE[8540] := 16#979A;
   // GBK_TO_UNICODE[8541] := 16#68DC;
   // GBK_TO_UNICODE[8542] := 16#979B;
   // GBK_TO_UNICODE[8543] := 16#68DD;
   // GBK_TO_UNICODE[8544] := 16#979C;
   // GBK_TO_UNICODE[8545] := 16#68DE;
   // GBK_TO_UNICODE[8546] := 16#979D;
   // GBK_TO_UNICODE[8547] := 16#68DF;
   // GBK_TO_UNICODE[8548] := 16#979E;
   // GBK_TO_UNICODE[8549] := 16#68E1;
   // GBK_TO_UNICODE[8550] := 16#979F;
   // GBK_TO_UNICODE[8551] := 16#68E2;
   // GBK_TO_UNICODE[8552] := 16#97A0;
   // GBK_TO_UNICODE[8553] := 16#68E4;
   // GBK_TO_UNICODE[8554] := 16#97A1;
   // GBK_TO_UNICODE[8555] := 16#68E5;
   // GBK_TO_UNICODE[8556] := 16#97A2;
   // GBK_TO_UNICODE[8557] := 16#68E6;
   // GBK_TO_UNICODE[8558] := 16#97A3;
   // GBK_TO_UNICODE[8559] := 16#68E7;
   // GBK_TO_UNICODE[8560] := 16#97A4;
   // GBK_TO_UNICODE[8561] := 16#68E8;
   // GBK_TO_UNICODE[8562] := 16#97A5;
   // GBK_TO_UNICODE[8563] := 16#68E9;
   // GBK_TO_UNICODE[8564] := 16#97A6;
   // GBK_TO_UNICODE[8565] := 16#68EA;
   // GBK_TO_UNICODE[8566] := 16#97A7;
   // GBK_TO_UNICODE[8567] := 16#68EB;
   // GBK_TO_UNICODE[8568] := 16#97A8;
   // GBK_TO_UNICODE[8569] := 16#68EC;
   // GBK_TO_UNICODE[8570] := 16#97A9;
   // GBK_TO_UNICODE[8571] := 16#68ED;
   // GBK_TO_UNICODE[8572] := 16#97AA;
   // GBK_TO_UNICODE[8573] := 16#68EF;
   // GBK_TO_UNICODE[8574] := 16#97AB;
   // GBK_TO_UNICODE[8575] := 16#68F2;
   // GBK_TO_UNICODE[8576] := 16#97AC;
   // GBK_TO_UNICODE[8577] := 16#68F3;
   // GBK_TO_UNICODE[8578] := 16#97AD;
   // GBK_TO_UNICODE[8579] := 16#68F4;
   // GBK_TO_UNICODE[8580] := 16#97AE;
   // GBK_TO_UNICODE[8581] := 16#68F6;
   // GBK_TO_UNICODE[8582] := 16#97AF;
   // GBK_TO_UNICODE[8583] := 16#68F7;
   // GBK_TO_UNICODE[8584] := 16#97B0;
   // GBK_TO_UNICODE[8585] := 16#68F8;
   // GBK_TO_UNICODE[8586] := 16#97B1;
   // GBK_TO_UNICODE[8587] := 16#68FB;
   // GBK_TO_UNICODE[8588] := 16#97B2;
   // GBK_TO_UNICODE[8589] := 16#68FD;
   // GBK_TO_UNICODE[8590] := 16#97B3;
   // GBK_TO_UNICODE[8591] := 16#68FE;
   // GBK_TO_UNICODE[8592] := 16#97B4;
   // GBK_TO_UNICODE[8593] := 16#68FF;
   // GBK_TO_UNICODE[8594] := 16#97B5;
   // GBK_TO_UNICODE[8595] := 16#6900;
   // GBK_TO_UNICODE[8596] := 16#97B6;
   // GBK_TO_UNICODE[8597] := 16#6902;
   // GBK_TO_UNICODE[8598] := 16#97B7;
   // GBK_TO_UNICODE[8599] := 16#6903;
   // GBK_TO_UNICODE[8600] := 16#97B8;
   // GBK_TO_UNICODE[8601] := 16#6904;
   // GBK_TO_UNICODE[8602] := 16#97B9;
   // GBK_TO_UNICODE[8603] := 16#6906;
   // GBK_TO_UNICODE[8604] := 16#97BA;
   // GBK_TO_UNICODE[8605] := 16#6907;
   // GBK_TO_UNICODE[8606] := 16#97BB;
   // GBK_TO_UNICODE[8607] := 16#6908;
   // GBK_TO_UNICODE[8608] := 16#97BC;
   // GBK_TO_UNICODE[8609] := 16#6909;
   // GBK_TO_UNICODE[8610] := 16#97BD;
   // GBK_TO_UNICODE[8611] := 16#690A;
   // GBK_TO_UNICODE[8612] := 16#97BE;
   // GBK_TO_UNICODE[8613] := 16#690C;
   // GBK_TO_UNICODE[8614] := 16#97BF;
   // GBK_TO_UNICODE[8615] := 16#690F;
   // GBK_TO_UNICODE[8616] := 16#97C0;
   // GBK_TO_UNICODE[8617] := 16#6911;
   // GBK_TO_UNICODE[8618] := 16#97C1;
   // GBK_TO_UNICODE[8619] := 16#6913;
   // GBK_TO_UNICODE[8620] := 16#97C2;
   // GBK_TO_UNICODE[8621] := 16#6914;
   // GBK_TO_UNICODE[8622] := 16#97C3;
   // GBK_TO_UNICODE[8623] := 16#6915;
   // GBK_TO_UNICODE[8624] := 16#97C4;
   // GBK_TO_UNICODE[8625] := 16#6916;
   // GBK_TO_UNICODE[8626] := 16#97C5;
   // GBK_TO_UNICODE[8627] := 16#6917;
   // GBK_TO_UNICODE[8628] := 16#97C6;
   // GBK_TO_UNICODE[8629] := 16#6918;
   // GBK_TO_UNICODE[8630] := 16#97C7;
   // GBK_TO_UNICODE[8631] := 16#6919;
   // GBK_TO_UNICODE[8632] := 16#97C8;
   // GBK_TO_UNICODE[8633] := 16#691A;
   // GBK_TO_UNICODE[8634] := 16#97C9;
   // GBK_TO_UNICODE[8635] := 16#691B;
   // GBK_TO_UNICODE[8636] := 16#97CA;
   // GBK_TO_UNICODE[8637] := 16#691C;
   // GBK_TO_UNICODE[8638] := 16#97CB;
   // GBK_TO_UNICODE[8639] := 16#691D;
   // GBK_TO_UNICODE[8640] := 16#97CC;
   // GBK_TO_UNICODE[8641] := 16#691E;
   // GBK_TO_UNICODE[8642] := 16#97CD;
   // GBK_TO_UNICODE[8643] := 16#6921;
   // GBK_TO_UNICODE[8644] := 16#97CE;
   // GBK_TO_UNICODE[8645] := 16#6922;
   // GBK_TO_UNICODE[8646] := 16#97CF;
   // GBK_TO_UNICODE[8647] := 16#6923;
   // GBK_TO_UNICODE[8648] := 16#97D0;
   // GBK_TO_UNICODE[8649] := 16#6925;
   // GBK_TO_UNICODE[8650] := 16#97D1;
   // GBK_TO_UNICODE[8651] := 16#6926;
   // GBK_TO_UNICODE[8652] := 16#97D2;
   // GBK_TO_UNICODE[8653] := 16#6927;
   // GBK_TO_UNICODE[8654] := 16#97D3;
   // GBK_TO_UNICODE[8655] := 16#6928;
   // GBK_TO_UNICODE[8656] := 16#97D4;
   // GBK_TO_UNICODE[8657] := 16#6929;
   // GBK_TO_UNICODE[8658] := 16#97D5;
   // GBK_TO_UNICODE[8659] := 16#692A;
   // GBK_TO_UNICODE[8660] := 16#97D6;
   // GBK_TO_UNICODE[8661] := 16#692B;
   // GBK_TO_UNICODE[8662] := 16#97D7;
   // GBK_TO_UNICODE[8663] := 16#692C;
   // GBK_TO_UNICODE[8664] := 16#97D8;
   // GBK_TO_UNICODE[8665] := 16#692E;
   // GBK_TO_UNICODE[8666] := 16#97D9;
   // GBK_TO_UNICODE[8667] := 16#692F;
   // GBK_TO_UNICODE[8668] := 16#97DA;
   // GBK_TO_UNICODE[8669] := 16#6931;
   // GBK_TO_UNICODE[8670] := 16#97DB;
   // GBK_TO_UNICODE[8671] := 16#6932;
   // GBK_TO_UNICODE[8672] := 16#97DC;
   // GBK_TO_UNICODE[8673] := 16#6933;
   // GBK_TO_UNICODE[8674] := 16#97DD;
   // GBK_TO_UNICODE[8675] := 16#6935;
   // GBK_TO_UNICODE[8676] := 16#97DE;
   // GBK_TO_UNICODE[8677] := 16#6936;
   // GBK_TO_UNICODE[8678] := 16#97DF;
   // GBK_TO_UNICODE[8679] := 16#6937;
   // GBK_TO_UNICODE[8680] := 16#97E0;
   // GBK_TO_UNICODE[8681] := 16#6938;
   // GBK_TO_UNICODE[8682] := 16#97E1;
   // GBK_TO_UNICODE[8683] := 16#693A;
   // GBK_TO_UNICODE[8684] := 16#97E2;
   // GBK_TO_UNICODE[8685] := 16#693B;
   // GBK_TO_UNICODE[8686] := 16#97E3;
   // GBK_TO_UNICODE[8687] := 16#693C;
   // GBK_TO_UNICODE[8688] := 16#97E4;
   // GBK_TO_UNICODE[8689] := 16#693E;
   // GBK_TO_UNICODE[8690] := 16#97E5;
   // GBK_TO_UNICODE[8691] := 16#6940;
   // GBK_TO_UNICODE[8692] := 16#97E6;
   // GBK_TO_UNICODE[8693] := 16#6941;
   // GBK_TO_UNICODE[8694] := 16#97E7;
   // GBK_TO_UNICODE[8695] := 16#6943;
   // GBK_TO_UNICODE[8696] := 16#97E8;
   // GBK_TO_UNICODE[8697] := 16#6944;
   // GBK_TO_UNICODE[8698] := 16#97E9;
   // GBK_TO_UNICODE[8699] := 16#6945;
   // GBK_TO_UNICODE[8700] := 16#97EA;
   // GBK_TO_UNICODE[8701] := 16#6946;
   // GBK_TO_UNICODE[8702] := 16#97EB;
   // GBK_TO_UNICODE[8703] := 16#6947;
   // GBK_TO_UNICODE[8704] := 16#97EC;
   // GBK_TO_UNICODE[8705] := 16#6948;
   // GBK_TO_UNICODE[8706] := 16#97ED;
   // GBK_TO_UNICODE[8707] := 16#6949;
   // GBK_TO_UNICODE[8708] := 16#97EE;
   // GBK_TO_UNICODE[8709] := 16#694A;
   // GBK_TO_UNICODE[8710] := 16#97EF;
   // GBK_TO_UNICODE[8711] := 16#694B;
   // GBK_TO_UNICODE[8712] := 16#97F0;
   // GBK_TO_UNICODE[8713] := 16#694C;
   // GBK_TO_UNICODE[8714] := 16#97F1;
   // GBK_TO_UNICODE[8715] := 16#694D;
   // GBK_TO_UNICODE[8716] := 16#97F2;
   // GBK_TO_UNICODE[8717] := 16#694E;
   // GBK_TO_UNICODE[8718] := 16#97F3;
   // GBK_TO_UNICODE[8719] := 16#694F;
   // GBK_TO_UNICODE[8720] := 16#97F4;
   // GBK_TO_UNICODE[8721] := 16#6950;
   // GBK_TO_UNICODE[8722] := 16#97F5;
   // GBK_TO_UNICODE[8723] := 16#6951;
   // GBK_TO_UNICODE[8724] := 16#97F6;
   // GBK_TO_UNICODE[8725] := 16#6952;
   // GBK_TO_UNICODE[8726] := 16#97F7;
   // GBK_TO_UNICODE[8727] := 16#6953;
   // GBK_TO_UNICODE[8728] := 16#97F8;
   // GBK_TO_UNICODE[8729] := 16#6955;
   // GBK_TO_UNICODE[8730] := 16#97F9;
   // GBK_TO_UNICODE[8731] := 16#6956;
   // GBK_TO_UNICODE[8732] := 16#97FA;
   // GBK_TO_UNICODE[8733] := 16#6958;
   // GBK_TO_UNICODE[8734] := 16#97FB;
   // GBK_TO_UNICODE[8735] := 16#6959;
   // GBK_TO_UNICODE[8736] := 16#97FC;
   // GBK_TO_UNICODE[8737] := 16#695B;
   // GBK_TO_UNICODE[8738] := 16#97FD;
   // GBK_TO_UNICODE[8739] := 16#695C;
   // GBK_TO_UNICODE[8740] := 16#97FE;
   // GBK_TO_UNICODE[8741] := 16#695F;
   // GBK_TO_UNICODE[8742] := 16#9840;
   // GBK_TO_UNICODE[8743] := 16#6961;
   // GBK_TO_UNICODE[8744] := 16#9841;
   // GBK_TO_UNICODE[8745] := 16#6962;
   // GBK_TO_UNICODE[8746] := 16#9842;
   // GBK_TO_UNICODE[8747] := 16#6964;
   // GBK_TO_UNICODE[8748] := 16#9843;
   // GBK_TO_UNICODE[8749] := 16#6965;
   // GBK_TO_UNICODE[8750] := 16#9844;
   // GBK_TO_UNICODE[8751] := 16#6967;
   // GBK_TO_UNICODE[8752] := 16#9845;
   // GBK_TO_UNICODE[8753] := 16#6968;
   // GBK_TO_UNICODE[8754] := 16#9846;
   // GBK_TO_UNICODE[8755] := 16#6969;
   // GBK_TO_UNICODE[8756] := 16#9847;
   // GBK_TO_UNICODE[8757] := 16#696A;
   // GBK_TO_UNICODE[8758] := 16#9848;
   // GBK_TO_UNICODE[8759] := 16#696C;
   // GBK_TO_UNICODE[8760] := 16#9849;
   // GBK_TO_UNICODE[8761] := 16#696D;
   // GBK_TO_UNICODE[8762] := 16#984A;
   // GBK_TO_UNICODE[8763] := 16#696F;
   // GBK_TO_UNICODE[8764] := 16#984B;
   // GBK_TO_UNICODE[8765] := 16#6970;
   // GBK_TO_UNICODE[8766] := 16#984C;
   // GBK_TO_UNICODE[8767] := 16#6972;
   // GBK_TO_UNICODE[8768] := 16#984D;
   // GBK_TO_UNICODE[8769] := 16#6973;
   // GBK_TO_UNICODE[8770] := 16#984E;
   // GBK_TO_UNICODE[8771] := 16#6974;
   // GBK_TO_UNICODE[8772] := 16#984F;
   // GBK_TO_UNICODE[8773] := 16#6975;
   // GBK_TO_UNICODE[8774] := 16#9850;
   // GBK_TO_UNICODE[8775] := 16#6976;
   // GBK_TO_UNICODE[8776] := 16#9851;
   // GBK_TO_UNICODE[8777] := 16#697A;
   // GBK_TO_UNICODE[8778] := 16#9852;
   // GBK_TO_UNICODE[8779] := 16#697B;
   // GBK_TO_UNICODE[8780] := 16#9853;
   // GBK_TO_UNICODE[8781] := 16#697D;
   // GBK_TO_UNICODE[8782] := 16#9854;
   // GBK_TO_UNICODE[8783] := 16#697E;
   // GBK_TO_UNICODE[8784] := 16#9855;
   // GBK_TO_UNICODE[8785] := 16#697F;
   // GBK_TO_UNICODE[8786] := 16#9856;
   // GBK_TO_UNICODE[8787] := 16#6981;
   // GBK_TO_UNICODE[8788] := 16#9857;
   // GBK_TO_UNICODE[8789] := 16#6983;
   // GBK_TO_UNICODE[8790] := 16#9858;
   // GBK_TO_UNICODE[8791] := 16#6985;
   // GBK_TO_UNICODE[8792] := 16#9859;
   // GBK_TO_UNICODE[8793] := 16#698A;
   // GBK_TO_UNICODE[8794] := 16#985A;
   // GBK_TO_UNICODE[8795] := 16#698B;
   // GBK_TO_UNICODE[8796] := 16#985B;
   // GBK_TO_UNICODE[8797] := 16#698C;
   // GBK_TO_UNICODE[8798] := 16#985C;
   // GBK_TO_UNICODE[8799] := 16#698E;
   // GBK_TO_UNICODE[8800] := 16#985D;
   // GBK_TO_UNICODE[8801] := 16#698F;
   // GBK_TO_UNICODE[8802] := 16#985E;
   // GBK_TO_UNICODE[8803] := 16#6990;
   // GBK_TO_UNICODE[8804] := 16#985F;
   // GBK_TO_UNICODE[8805] := 16#6991;
   // GBK_TO_UNICODE[8806] := 16#9860;
   // GBK_TO_UNICODE[8807] := 16#6992;
   // GBK_TO_UNICODE[8808] := 16#9861;
   // GBK_TO_UNICODE[8809] := 16#6993;
   // GBK_TO_UNICODE[8810] := 16#9862;
   // GBK_TO_UNICODE[8811] := 16#6996;
   // GBK_TO_UNICODE[8812] := 16#9863;
   // GBK_TO_UNICODE[8813] := 16#6997;
   // GBK_TO_UNICODE[8814] := 16#9864;
   // GBK_TO_UNICODE[8815] := 16#6999;
   // GBK_TO_UNICODE[8816] := 16#9865;
   // GBK_TO_UNICODE[8817] := 16#699A;
   // GBK_TO_UNICODE[8818] := 16#9866;
   // GBK_TO_UNICODE[8819] := 16#699D;
   // GBK_TO_UNICODE[8820] := 16#9867;
   // GBK_TO_UNICODE[8821] := 16#699E;
   // GBK_TO_UNICODE[8822] := 16#9868;
   // GBK_TO_UNICODE[8823] := 16#699F;
   // GBK_TO_UNICODE[8824] := 16#9869;
   // GBK_TO_UNICODE[8825] := 16#69A0;
   // GBK_TO_UNICODE[8826] := 16#986A;
   // GBK_TO_UNICODE[8827] := 16#69A1;
   // GBK_TO_UNICODE[8828] := 16#986B;
   // GBK_TO_UNICODE[8829] := 16#69A2;
   // GBK_TO_UNICODE[8830] := 16#986C;
   // GBK_TO_UNICODE[8831] := 16#69A3;
   // GBK_TO_UNICODE[8832] := 16#986D;
   // GBK_TO_UNICODE[8833] := 16#69A4;
   // GBK_TO_UNICODE[8834] := 16#986E;
   // GBK_TO_UNICODE[8835] := 16#69A5;
   // GBK_TO_UNICODE[8836] := 16#986F;
   // GBK_TO_UNICODE[8837] := 16#69A6;
   // GBK_TO_UNICODE[8838] := 16#9870;
   // GBK_TO_UNICODE[8839] := 16#69A9;
   // GBK_TO_UNICODE[8840] := 16#9871;
   // GBK_TO_UNICODE[8841] := 16#69AA;
   // GBK_TO_UNICODE[8842] := 16#9872;
   // GBK_TO_UNICODE[8843] := 16#69AC;
   // GBK_TO_UNICODE[8844] := 16#9873;
   // GBK_TO_UNICODE[8845] := 16#69AE;
   // GBK_TO_UNICODE[8846] := 16#9874;
   // GBK_TO_UNICODE[8847] := 16#69AF;
   // GBK_TO_UNICODE[8848] := 16#9875;
   // GBK_TO_UNICODE[8849] := 16#69B0;
   // GBK_TO_UNICODE[8850] := 16#9876;
   // GBK_TO_UNICODE[8851] := 16#69B2;
   // GBK_TO_UNICODE[8852] := 16#9877;
   // GBK_TO_UNICODE[8853] := 16#69B3;
   // GBK_TO_UNICODE[8854] := 16#9878;
   // GBK_TO_UNICODE[8855] := 16#69B5;
   // GBK_TO_UNICODE[8856] := 16#9879;
   // GBK_TO_UNICODE[8857] := 16#69B6;
   // GBK_TO_UNICODE[8858] := 16#987A;
   // GBK_TO_UNICODE[8859] := 16#69B8;
   // GBK_TO_UNICODE[8860] := 16#987B;
   // GBK_TO_UNICODE[8861] := 16#69B9;
   // GBK_TO_UNICODE[8862] := 16#987C;
   // GBK_TO_UNICODE[8863] := 16#69BA;
   // GBK_TO_UNICODE[8864] := 16#987D;
   // GBK_TO_UNICODE[8865] := 16#69BC;
   // GBK_TO_UNICODE[8866] := 16#987E;
   // GBK_TO_UNICODE[8867] := 16#69BD;
   // GBK_TO_UNICODE[8868] := 16#9880;
   // GBK_TO_UNICODE[8869] := 16#69BE;
   // GBK_TO_UNICODE[8870] := 16#9881;
   // GBK_TO_UNICODE[8871] := 16#69BF;
   // GBK_TO_UNICODE[8872] := 16#9882;
   // GBK_TO_UNICODE[8873] := 16#69C0;
   // GBK_TO_UNICODE[8874] := 16#9883;
   // GBK_TO_UNICODE[8875] := 16#69C2;
   // GBK_TO_UNICODE[8876] := 16#9884;
   // GBK_TO_UNICODE[8877] := 16#69C3;
   // GBK_TO_UNICODE[8878] := 16#9885;
   // GBK_TO_UNICODE[8879] := 16#69C4;
   // GBK_TO_UNICODE[8880] := 16#9886;
   // GBK_TO_UNICODE[8881] := 16#69C5;
   // GBK_TO_UNICODE[8882] := 16#9887;
   // GBK_TO_UNICODE[8883] := 16#69C6;
   // GBK_TO_UNICODE[8884] := 16#9888;
   // GBK_TO_UNICODE[8885] := 16#69C7;
   // GBK_TO_UNICODE[8886] := 16#9889;
   // GBK_TO_UNICODE[8887] := 16#69C8;
   // GBK_TO_UNICODE[8888] := 16#988A;
   // GBK_TO_UNICODE[8889] := 16#69C9;
   // GBK_TO_UNICODE[8890] := 16#988B;
   // GBK_TO_UNICODE[8891] := 16#69CB;
   // GBK_TO_UNICODE[8892] := 16#988C;
   // GBK_TO_UNICODE[8893] := 16#69CD;
   // GBK_TO_UNICODE[8894] := 16#988D;
   // GBK_TO_UNICODE[8895] := 16#69CF;
   // GBK_TO_UNICODE[8896] := 16#988E;
   // GBK_TO_UNICODE[8897] := 16#69D1;
   // GBK_TO_UNICODE[8898] := 16#988F;
   // GBK_TO_UNICODE[8899] := 16#69D2;
   // GBK_TO_UNICODE[8900] := 16#9890;
   // GBK_TO_UNICODE[8901] := 16#69D3;
   // GBK_TO_UNICODE[8902] := 16#9891;
   // GBK_TO_UNICODE[8903] := 16#69D5;
   // GBK_TO_UNICODE[8904] := 16#9892;
   // GBK_TO_UNICODE[8905] := 16#69D6;
   // GBK_TO_UNICODE[8906] := 16#9893;
   // GBK_TO_UNICODE[8907] := 16#69D7;
   // GBK_TO_UNICODE[8908] := 16#9894;
   // GBK_TO_UNICODE[8909] := 16#69D8;
   // GBK_TO_UNICODE[8910] := 16#9895;
   // GBK_TO_UNICODE[8911] := 16#69D9;
   // GBK_TO_UNICODE[8912] := 16#9896;
   // GBK_TO_UNICODE[8913] := 16#69DA;
   // GBK_TO_UNICODE[8914] := 16#9897;
   // GBK_TO_UNICODE[8915] := 16#69DC;
   // GBK_TO_UNICODE[8916] := 16#9898;
   // GBK_TO_UNICODE[8917] := 16#69DD;
   // GBK_TO_UNICODE[8918] := 16#9899;
   // GBK_TO_UNICODE[8919] := 16#69DE;
   // GBK_TO_UNICODE[8920] := 16#989A;
   // GBK_TO_UNICODE[8921] := 16#69E1;
   // GBK_TO_UNICODE[8922] := 16#989B;
   // GBK_TO_UNICODE[8923] := 16#69E2;
   // GBK_TO_UNICODE[8924] := 16#989C;
   // GBK_TO_UNICODE[8925] := 16#69E3;
   // GBK_TO_UNICODE[8926] := 16#989D;
   // GBK_TO_UNICODE[8927] := 16#69E4;
   // GBK_TO_UNICODE[8928] := 16#989E;
   // GBK_TO_UNICODE[8929] := 16#69E5;
   // GBK_TO_UNICODE[8930] := 16#989F;
   // GBK_TO_UNICODE[8931] := 16#69E6;
   // GBK_TO_UNICODE[8932] := 16#98A0;
   // GBK_TO_UNICODE[8933] := 16#69E7;
   // GBK_TO_UNICODE[8934] := 16#98A1;
   // GBK_TO_UNICODE[8935] := 16#69E8;
   // GBK_TO_UNICODE[8936] := 16#98A2;
   // GBK_TO_UNICODE[8937] := 16#69E9;
   // GBK_TO_UNICODE[8938] := 16#98A3;
   // GBK_TO_UNICODE[8939] := 16#69EA;
   // GBK_TO_UNICODE[8940] := 16#98A4;
   // GBK_TO_UNICODE[8941] := 16#69EB;
   // GBK_TO_UNICODE[8942] := 16#98A5;
   // GBK_TO_UNICODE[8943] := 16#69EC;
   // GBK_TO_UNICODE[8944] := 16#98A6;
   // GBK_TO_UNICODE[8945] := 16#69EE;
   // GBK_TO_UNICODE[8946] := 16#98A7;
   // GBK_TO_UNICODE[8947] := 16#69EF;
   // GBK_TO_UNICODE[8948] := 16#98A8;
   // GBK_TO_UNICODE[8949] := 16#69F0;
   // GBK_TO_UNICODE[8950] := 16#98A9;
   // GBK_TO_UNICODE[8951] := 16#69F1;
   // GBK_TO_UNICODE[8952] := 16#98AA;
   // GBK_TO_UNICODE[8953] := 16#69F3;
   // GBK_TO_UNICODE[8954] := 16#98AB;
   // GBK_TO_UNICODE[8955] := 16#69F4;
   // GBK_TO_UNICODE[8956] := 16#98AC;
   // GBK_TO_UNICODE[8957] := 16#69F5;
   // GBK_TO_UNICODE[8958] := 16#98AD;
   // GBK_TO_UNICODE[8959] := 16#69F6;
   // GBK_TO_UNICODE[8960] := 16#98AE;
   // GBK_TO_UNICODE[8961] := 16#69F7;
   // GBK_TO_UNICODE[8962] := 16#98AF;
   // GBK_TO_UNICODE[8963] := 16#69F8;
   // GBK_TO_UNICODE[8964] := 16#98B0;
   // GBK_TO_UNICODE[8965] := 16#69F9;
   // GBK_TO_UNICODE[8966] := 16#98B1;
   // GBK_TO_UNICODE[8967] := 16#69FA;
   // GBK_TO_UNICODE[8968] := 16#98B2;
   // GBK_TO_UNICODE[8969] := 16#69FB;
   // GBK_TO_UNICODE[8970] := 16#98B3;
   // GBK_TO_UNICODE[8971] := 16#69FC;
   // GBK_TO_UNICODE[8972] := 16#98B4;
   // GBK_TO_UNICODE[8973] := 16#69FE;
   // GBK_TO_UNICODE[8974] := 16#98B5;
   // GBK_TO_UNICODE[8975] := 16#6A00;
   // GBK_TO_UNICODE[8976] := 16#98B6;
   // GBK_TO_UNICODE[8977] := 16#6A01;
   // GBK_TO_UNICODE[8978] := 16#98B7;
   // GBK_TO_UNICODE[8979] := 16#6A02;
   // GBK_TO_UNICODE[8980] := 16#98B8;
   // GBK_TO_UNICODE[8981] := 16#6A03;
   // GBK_TO_UNICODE[8982] := 16#98B9;
   // GBK_TO_UNICODE[8983] := 16#6A04;
   // GBK_TO_UNICODE[8984] := 16#98BA;
   // GBK_TO_UNICODE[8985] := 16#6A05;
   // GBK_TO_UNICODE[8986] := 16#98BB;
   // GBK_TO_UNICODE[8987] := 16#6A06;
   // GBK_TO_UNICODE[8988] := 16#98BC;
   // GBK_TO_UNICODE[8989] := 16#6A07;
   // GBK_TO_UNICODE[8990] := 16#98BD;
   // GBK_TO_UNICODE[8991] := 16#6A08;
   // GBK_TO_UNICODE[8992] := 16#98BE;
   // GBK_TO_UNICODE[8993] := 16#6A09;
   // GBK_TO_UNICODE[8994] := 16#98BF;
   // GBK_TO_UNICODE[8995] := 16#6A0B;
   // GBK_TO_UNICODE[8996] := 16#98C0;
   // GBK_TO_UNICODE[8997] := 16#6A0C;
   // GBK_TO_UNICODE[8998] := 16#98C1;
   // GBK_TO_UNICODE[8999] := 16#6A0D;
   // GBK_TO_UNICODE[9000] := 16#98C2;
   // GBK_TO_UNICODE[9001] := 16#6A0E;
   // GBK_TO_UNICODE[9002] := 16#98C3;
   // GBK_TO_UNICODE[9003] := 16#6A0F;
   // GBK_TO_UNICODE[9004] := 16#98C4;
   // GBK_TO_UNICODE[9005] := 16#6A10;
   // GBK_TO_UNICODE[9006] := 16#98C5;
   // GBK_TO_UNICODE[9007] := 16#6A11;
   // GBK_TO_UNICODE[9008] := 16#98C6;
   // GBK_TO_UNICODE[9009] := 16#6A12;
   // GBK_TO_UNICODE[9010] := 16#98C7;
   // GBK_TO_UNICODE[9011] := 16#6A13;
   // GBK_TO_UNICODE[9012] := 16#98C8;
   // GBK_TO_UNICODE[9013] := 16#6A14;
   // GBK_TO_UNICODE[9014] := 16#98C9;
   // GBK_TO_UNICODE[9015] := 16#6A15;
   // GBK_TO_UNICODE[9016] := 16#98CA;
   // GBK_TO_UNICODE[9017] := 16#6A16;
   // GBK_TO_UNICODE[9018] := 16#98CB;
   // GBK_TO_UNICODE[9019] := 16#6A19;
   // GBK_TO_UNICODE[9020] := 16#98CC;
   // GBK_TO_UNICODE[9021] := 16#6A1A;
   // GBK_TO_UNICODE[9022] := 16#98CD;
   // GBK_TO_UNICODE[9023] := 16#6A1B;
   // GBK_TO_UNICODE[9024] := 16#98CE;
   // GBK_TO_UNICODE[9025] := 16#6A1C;
   // GBK_TO_UNICODE[9026] := 16#98CF;
   // GBK_TO_UNICODE[9027] := 16#6A1D;
   // GBK_TO_UNICODE[9028] := 16#98D0;
   // GBK_TO_UNICODE[9029] := 16#6A1E;
   // GBK_TO_UNICODE[9030] := 16#98D1;
   // GBK_TO_UNICODE[9031] := 16#6A20;
   // GBK_TO_UNICODE[9032] := 16#98D2;
   // GBK_TO_UNICODE[9033] := 16#6A22;
   // GBK_TO_UNICODE[9034] := 16#98D3;
   // GBK_TO_UNICODE[9035] := 16#6A23;
   // GBK_TO_UNICODE[9036] := 16#98D4;
   // GBK_TO_UNICODE[9037] := 16#6A24;
   // GBK_TO_UNICODE[9038] := 16#98D5;
   // GBK_TO_UNICODE[9039] := 16#6A25;
   // GBK_TO_UNICODE[9040] := 16#98D6;
   // GBK_TO_UNICODE[9041] := 16#6A26;
   // GBK_TO_UNICODE[9042] := 16#98D7;
   // GBK_TO_UNICODE[9043] := 16#6A27;
   // GBK_TO_UNICODE[9044] := 16#98D8;
   // GBK_TO_UNICODE[9045] := 16#6A29;
   // GBK_TO_UNICODE[9046] := 16#98D9;
   // GBK_TO_UNICODE[9047] := 16#6A2B;
   // GBK_TO_UNICODE[9048] := 16#98DA;
   // GBK_TO_UNICODE[9049] := 16#6A2C;
   // GBK_TO_UNICODE[9050] := 16#98DB;
   // GBK_TO_UNICODE[9051] := 16#6A2D;
   // GBK_TO_UNICODE[9052] := 16#98DC;
   // GBK_TO_UNICODE[9053] := 16#6A2E;
   // GBK_TO_UNICODE[9054] := 16#98DD;
   // GBK_TO_UNICODE[9055] := 16#6A30;
   // GBK_TO_UNICODE[9056] := 16#98DE;
   // GBK_TO_UNICODE[9057] := 16#6A32;
   // GBK_TO_UNICODE[9058] := 16#98DF;
   // GBK_TO_UNICODE[9059] := 16#6A33;
   // GBK_TO_UNICODE[9060] := 16#98E0;
   // GBK_TO_UNICODE[9061] := 16#6A34;
   // GBK_TO_UNICODE[9062] := 16#98E1;
   // GBK_TO_UNICODE[9063] := 16#6A36;
   // GBK_TO_UNICODE[9064] := 16#98E2;
   // GBK_TO_UNICODE[9065] := 16#6A37;
   // GBK_TO_UNICODE[9066] := 16#98E3;
   // GBK_TO_UNICODE[9067] := 16#6A38;
   // GBK_TO_UNICODE[9068] := 16#98E4;
   // GBK_TO_UNICODE[9069] := 16#6A39;
   // GBK_TO_UNICODE[9070] := 16#98E5;
   // GBK_TO_UNICODE[9071] := 16#6A3A;
   // GBK_TO_UNICODE[9072] := 16#98E6;
   // GBK_TO_UNICODE[9073] := 16#6A3B;
   // GBK_TO_UNICODE[9074] := 16#98E7;
   // GBK_TO_UNICODE[9075] := 16#6A3C;
   // GBK_TO_UNICODE[9076] := 16#98E8;
   // GBK_TO_UNICODE[9077] := 16#6A3F;
   // GBK_TO_UNICODE[9078] := 16#98E9;
   // GBK_TO_UNICODE[9079] := 16#6A40;
   // GBK_TO_UNICODE[9080] := 16#98EA;
   // GBK_TO_UNICODE[9081] := 16#6A41;
   // GBK_TO_UNICODE[9082] := 16#98EB;
   // GBK_TO_UNICODE[9083] := 16#6A42;
   // GBK_TO_UNICODE[9084] := 16#98EC;
   // GBK_TO_UNICODE[9085] := 16#6A43;
   // GBK_TO_UNICODE[9086] := 16#98ED;
   // GBK_TO_UNICODE[9087] := 16#6A45;
   // GBK_TO_UNICODE[9088] := 16#98EE;
   // GBK_TO_UNICODE[9089] := 16#6A46;
   // GBK_TO_UNICODE[9090] := 16#98EF;
   // GBK_TO_UNICODE[9091] := 16#6A48;
   // GBK_TO_UNICODE[9092] := 16#98F0;
   // GBK_TO_UNICODE[9093] := 16#6A49;
   // GBK_TO_UNICODE[9094] := 16#98F1;
   // GBK_TO_UNICODE[9095] := 16#6A4A;
   // GBK_TO_UNICODE[9096] := 16#98F2;
   // GBK_TO_UNICODE[9097] := 16#6A4B;
   // GBK_TO_UNICODE[9098] := 16#98F3;
   // GBK_TO_UNICODE[9099] := 16#6A4C;
   // GBK_TO_UNICODE[9100] := 16#98F4;
   // GBK_TO_UNICODE[9101] := 16#6A4D;
   // GBK_TO_UNICODE[9102] := 16#98F5;
   // GBK_TO_UNICODE[9103] := 16#6A4E;
   // GBK_TO_UNICODE[9104] := 16#98F6;
   // GBK_TO_UNICODE[9105] := 16#6A4F;
   // GBK_TO_UNICODE[9106] := 16#98F7;
   // GBK_TO_UNICODE[9107] := 16#6A51;
   // GBK_TO_UNICODE[9108] := 16#98F8;
   // GBK_TO_UNICODE[9109] := 16#6A52;
   // GBK_TO_UNICODE[9110] := 16#98F9;
   // GBK_TO_UNICODE[9111] := 16#6A53;
   // GBK_TO_UNICODE[9112] := 16#98FA;
   // GBK_TO_UNICODE[9113] := 16#6A54;
   // GBK_TO_UNICODE[9114] := 16#98FB;
   // GBK_TO_UNICODE[9115] := 16#6A55;
   // GBK_TO_UNICODE[9116] := 16#98FC;
   // GBK_TO_UNICODE[9117] := 16#6A56;
   // GBK_TO_UNICODE[9118] := 16#98FD;
   // GBK_TO_UNICODE[9119] := 16#6A57;
   // GBK_TO_UNICODE[9120] := 16#98FE;
   // GBK_TO_UNICODE[9121] := 16#6A5A;
   // GBK_TO_UNICODE[9122] := 16#9940;
   // GBK_TO_UNICODE[9123] := 16#6A5C;
   // GBK_TO_UNICODE[9124] := 16#9941;
   // GBK_TO_UNICODE[9125] := 16#6A5D;
   // GBK_TO_UNICODE[9126] := 16#9942;
   // GBK_TO_UNICODE[9127] := 16#6A5E;
   // GBK_TO_UNICODE[9128] := 16#9943;
   // GBK_TO_UNICODE[9129] := 16#6A5F;
   // GBK_TO_UNICODE[9130] := 16#9944;
   // GBK_TO_UNICODE[9131] := 16#6A60;
   // GBK_TO_UNICODE[9132] := 16#9945;
   // GBK_TO_UNICODE[9133] := 16#6A62;
   // GBK_TO_UNICODE[9134] := 16#9946;
   // GBK_TO_UNICODE[9135] := 16#6A63;
   // GBK_TO_UNICODE[9136] := 16#9947;
   // GBK_TO_UNICODE[9137] := 16#6A64;
   // GBK_TO_UNICODE[9138] := 16#9948;
   // GBK_TO_UNICODE[9139] := 16#6A66;
   // GBK_TO_UNICODE[9140] := 16#9949;
   // GBK_TO_UNICODE[9141] := 16#6A67;
   // GBK_TO_UNICODE[9142] := 16#994A;
   // GBK_TO_UNICODE[9143] := 16#6A68;
   // GBK_TO_UNICODE[9144] := 16#994B;
   // GBK_TO_UNICODE[9145] := 16#6A69;
   // GBK_TO_UNICODE[9146] := 16#994C;
   // GBK_TO_UNICODE[9147] := 16#6A6A;
   // GBK_TO_UNICODE[9148] := 16#994D;
   // GBK_TO_UNICODE[9149] := 16#6A6B;
   // GBK_TO_UNICODE[9150] := 16#994E;
   // GBK_TO_UNICODE[9151] := 16#6A6C;
   // GBK_TO_UNICODE[9152] := 16#994F;
   // GBK_TO_UNICODE[9153] := 16#6A6D;
   // GBK_TO_UNICODE[9154] := 16#9950;
   // GBK_TO_UNICODE[9155] := 16#6A6E;
   // GBK_TO_UNICODE[9156] := 16#9951;
   // GBK_TO_UNICODE[9157] := 16#6A6F;
   // GBK_TO_UNICODE[9158] := 16#9952;
   // GBK_TO_UNICODE[9159] := 16#6A70;
   // GBK_TO_UNICODE[9160] := 16#9953;
   // GBK_TO_UNICODE[9161] := 16#6A72;
   // GBK_TO_UNICODE[9162] := 16#9954;
   // GBK_TO_UNICODE[9163] := 16#6A73;
   // GBK_TO_UNICODE[9164] := 16#9955;
   // GBK_TO_UNICODE[9165] := 16#6A74;
   // GBK_TO_UNICODE[9166] := 16#9956;
   // GBK_TO_UNICODE[9167] := 16#6A75;
   // GBK_TO_UNICODE[9168] := 16#9957;
   // GBK_TO_UNICODE[9169] := 16#6A76;
   // GBK_TO_UNICODE[9170] := 16#9958;
   // GBK_TO_UNICODE[9171] := 16#6A77;
   // GBK_TO_UNICODE[9172] := 16#9959;
   // GBK_TO_UNICODE[9173] := 16#6A78;
   // GBK_TO_UNICODE[9174] := 16#995A;
   // GBK_TO_UNICODE[9175] := 16#6A7A;
   // GBK_TO_UNICODE[9176] := 16#995B;
   // GBK_TO_UNICODE[9177] := 16#6A7B;
   // GBK_TO_UNICODE[9178] := 16#995C;
   // GBK_TO_UNICODE[9179] := 16#6A7D;
   // GBK_TO_UNICODE[9180] := 16#995D;
   // GBK_TO_UNICODE[9181] := 16#6A7E;
   // GBK_TO_UNICODE[9182] := 16#995E;
   // GBK_TO_UNICODE[9183] := 16#6A7F;
   // GBK_TO_UNICODE[9184] := 16#995F;
   // GBK_TO_UNICODE[9185] := 16#6A81;
   // GBK_TO_UNICODE[9186] := 16#9960;
   // GBK_TO_UNICODE[9187] := 16#6A82;
   // GBK_TO_UNICODE[9188] := 16#9961;
   // GBK_TO_UNICODE[9189] := 16#6A83;
   // GBK_TO_UNICODE[9190] := 16#9962;
   // GBK_TO_UNICODE[9191] := 16#6A85;
   // GBK_TO_UNICODE[9192] := 16#9963;
   // GBK_TO_UNICODE[9193] := 16#6A86;
   // GBK_TO_UNICODE[9194] := 16#9964;
   // GBK_TO_UNICODE[9195] := 16#6A87;
   // GBK_TO_UNICODE[9196] := 16#9965;
   // GBK_TO_UNICODE[9197] := 16#6A88;
   // GBK_TO_UNICODE[9198] := 16#9966;
   // GBK_TO_UNICODE[9199] := 16#6A89;
   // GBK_TO_UNICODE[9200] := 16#9967;
   // GBK_TO_UNICODE[9201] := 16#6A8A;
   // GBK_TO_UNICODE[9202] := 16#9968;
   // GBK_TO_UNICODE[9203] := 16#6A8B;
   // GBK_TO_UNICODE[9204] := 16#9969;
   // GBK_TO_UNICODE[9205] := 16#6A8C;
   // GBK_TO_UNICODE[9206] := 16#996A;
   // GBK_TO_UNICODE[9207] := 16#6A8D;
   // GBK_TO_UNICODE[9208] := 16#996B;
   // GBK_TO_UNICODE[9209] := 16#6A8F;
   // GBK_TO_UNICODE[9210] := 16#996C;
   // GBK_TO_UNICODE[9211] := 16#6A92;
   // GBK_TO_UNICODE[9212] := 16#996D;
   // GBK_TO_UNICODE[9213] := 16#6A93;
   // GBK_TO_UNICODE[9214] := 16#996E;
   // GBK_TO_UNICODE[9215] := 16#6A94;
   // GBK_TO_UNICODE[9216] := 16#996F;
   // GBK_TO_UNICODE[9217] := 16#6A95;
   // GBK_TO_UNICODE[9218] := 16#9970;
   // GBK_TO_UNICODE[9219] := 16#6A96;
   // GBK_TO_UNICODE[9220] := 16#9971;
   // GBK_TO_UNICODE[9221] := 16#6A98;
   // GBK_TO_UNICODE[9222] := 16#9972;
   // GBK_TO_UNICODE[9223] := 16#6A99;
   // GBK_TO_UNICODE[9224] := 16#9973;
   // GBK_TO_UNICODE[9225] := 16#6A9A;
   // GBK_TO_UNICODE[9226] := 16#9974;
   // GBK_TO_UNICODE[9227] := 16#6A9B;
   // GBK_TO_UNICODE[9228] := 16#9975;
   // GBK_TO_UNICODE[9229] := 16#6A9C;
   // GBK_TO_UNICODE[9230] := 16#9976;
   // GBK_TO_UNICODE[9231] := 16#6A9D;
   // GBK_TO_UNICODE[9232] := 16#9977;
   // GBK_TO_UNICODE[9233] := 16#6A9E;
   // GBK_TO_UNICODE[9234] := 16#9978;
   // GBK_TO_UNICODE[9235] := 16#6A9F;
   // GBK_TO_UNICODE[9236] := 16#9979;
   // GBK_TO_UNICODE[9237] := 16#6AA1;
   // GBK_TO_UNICODE[9238] := 16#997A;
   // GBK_TO_UNICODE[9239] := 16#6AA2;
   // GBK_TO_UNICODE[9240] := 16#997B;
   // GBK_TO_UNICODE[9241] := 16#6AA3;
   // GBK_TO_UNICODE[9242] := 16#997C;
   // GBK_TO_UNICODE[9243] := 16#6AA4;
   // GBK_TO_UNICODE[9244] := 16#997D;
   // GBK_TO_UNICODE[9245] := 16#6AA5;
   // GBK_TO_UNICODE[9246] := 16#997E;
   // GBK_TO_UNICODE[9247] := 16#6AA6;
   // GBK_TO_UNICODE[9248] := 16#9980;
   // GBK_TO_UNICODE[9249] := 16#6AA7;
   // GBK_TO_UNICODE[9250] := 16#9981;
   // GBK_TO_UNICODE[9251] := 16#6AA8;
   // GBK_TO_UNICODE[9252] := 16#9982;
   // GBK_TO_UNICODE[9253] := 16#6AAA;
   // GBK_TO_UNICODE[9254] := 16#9983;
   // GBK_TO_UNICODE[9255] := 16#6AAD;
   // GBK_TO_UNICODE[9256] := 16#9984;
   // GBK_TO_UNICODE[9257] := 16#6AAE;
   // GBK_TO_UNICODE[9258] := 16#9985;
   // GBK_TO_UNICODE[9259] := 16#6AAF;
   // GBK_TO_UNICODE[9260] := 16#9986;
   // GBK_TO_UNICODE[9261] := 16#6AB0;
   // GBK_TO_UNICODE[9262] := 16#9987;
   // GBK_TO_UNICODE[9263] := 16#6AB1;
   // GBK_TO_UNICODE[9264] := 16#9988;
   // GBK_TO_UNICODE[9265] := 16#6AB2;
   // GBK_TO_UNICODE[9266] := 16#9989;
   // GBK_TO_UNICODE[9267] := 16#6AB3;
   // GBK_TO_UNICODE[9268] := 16#998A;
   // GBK_TO_UNICODE[9269] := 16#6AB4;
   // GBK_TO_UNICODE[9270] := 16#998B;
   // GBK_TO_UNICODE[9271] := 16#6AB5;
   // GBK_TO_UNICODE[9272] := 16#998C;
   // GBK_TO_UNICODE[9273] := 16#6AB6;
   // GBK_TO_UNICODE[9274] := 16#998D;
   // GBK_TO_UNICODE[9275] := 16#6AB7;
   // GBK_TO_UNICODE[9276] := 16#998E;
   // GBK_TO_UNICODE[9277] := 16#6AB8;
   // GBK_TO_UNICODE[9278] := 16#998F;
   // GBK_TO_UNICODE[9279] := 16#6AB9;
   // GBK_TO_UNICODE[9280] := 16#9990;
   // GBK_TO_UNICODE[9281] := 16#6ABA;
   // GBK_TO_UNICODE[9282] := 16#9991;
   // GBK_TO_UNICODE[9283] := 16#6ABB;
   // GBK_TO_UNICODE[9284] := 16#9992;
   // GBK_TO_UNICODE[9285] := 16#6ABC;
   // GBK_TO_UNICODE[9286] := 16#9993;
   // GBK_TO_UNICODE[9287] := 16#6ABD;
   // GBK_TO_UNICODE[9288] := 16#9994;
   // GBK_TO_UNICODE[9289] := 16#6ABE;
   // GBK_TO_UNICODE[9290] := 16#9995;
   // GBK_TO_UNICODE[9291] := 16#6ABF;
   // GBK_TO_UNICODE[9292] := 16#9996;
   // GBK_TO_UNICODE[9293] := 16#6AC0;
   // GBK_TO_UNICODE[9294] := 16#9997;
   // GBK_TO_UNICODE[9295] := 16#6AC1;
   // GBK_TO_UNICODE[9296] := 16#9998;
   // GBK_TO_UNICODE[9297] := 16#6AC2;
   // GBK_TO_UNICODE[9298] := 16#9999;
   // GBK_TO_UNICODE[9299] := 16#6AC3;
   // GBK_TO_UNICODE[9300] := 16#999A;
   // GBK_TO_UNICODE[9301] := 16#6AC4;
   // GBK_TO_UNICODE[9302] := 16#999B;
   // GBK_TO_UNICODE[9303] := 16#6AC5;
   // GBK_TO_UNICODE[9304] := 16#999C;
   // GBK_TO_UNICODE[9305] := 16#6AC6;
   // GBK_TO_UNICODE[9306] := 16#999D;
   // GBK_TO_UNICODE[9307] := 16#6AC7;
   // GBK_TO_UNICODE[9308] := 16#999E;
   // GBK_TO_UNICODE[9309] := 16#6AC8;
   // GBK_TO_UNICODE[9310] := 16#999F;
   // GBK_TO_UNICODE[9311] := 16#6AC9;
   // GBK_TO_UNICODE[9312] := 16#99A0;
   // GBK_TO_UNICODE[9313] := 16#6ACA;
   // GBK_TO_UNICODE[9314] := 16#99A1;
   // GBK_TO_UNICODE[9315] := 16#6ACB;
   // GBK_TO_UNICODE[9316] := 16#99A2;
   // GBK_TO_UNICODE[9317] := 16#6ACC;
   // GBK_TO_UNICODE[9318] := 16#99A3;
   // GBK_TO_UNICODE[9319] := 16#6ACD;
   // GBK_TO_UNICODE[9320] := 16#99A4;
   // GBK_TO_UNICODE[9321] := 16#6ACE;
   // GBK_TO_UNICODE[9322] := 16#99A5;
   // GBK_TO_UNICODE[9323] := 16#6ACF;
   // GBK_TO_UNICODE[9324] := 16#99A6;
   // GBK_TO_UNICODE[9325] := 16#6AD0;
   // GBK_TO_UNICODE[9326] := 16#99A7;
   // GBK_TO_UNICODE[9327] := 16#6AD1;
   // GBK_TO_UNICODE[9328] := 16#99A8;
   // GBK_TO_UNICODE[9329] := 16#6AD2;
   // GBK_TO_UNICODE[9330] := 16#99A9;
   // GBK_TO_UNICODE[9331] := 16#6AD3;
   // GBK_TO_UNICODE[9332] := 16#99AA;
   // GBK_TO_UNICODE[9333] := 16#6AD4;
   // GBK_TO_UNICODE[9334] := 16#99AB;
   // GBK_TO_UNICODE[9335] := 16#6AD5;
   // GBK_TO_UNICODE[9336] := 16#99AC;
   // GBK_TO_UNICODE[9337] := 16#6AD6;
   // GBK_TO_UNICODE[9338] := 16#99AD;
   // GBK_TO_UNICODE[9339] := 16#6AD7;
   // GBK_TO_UNICODE[9340] := 16#99AE;
   // GBK_TO_UNICODE[9341] := 16#6AD8;
   // GBK_TO_UNICODE[9342] := 16#99AF;
   // GBK_TO_UNICODE[9343] := 16#6AD9;
   // GBK_TO_UNICODE[9344] := 16#99B0;
   // GBK_TO_UNICODE[9345] := 16#6ADA;
   // GBK_TO_UNICODE[9346] := 16#99B1;
   // GBK_TO_UNICODE[9347] := 16#6ADB;
   // GBK_TO_UNICODE[9348] := 16#99B2;
   // GBK_TO_UNICODE[9349] := 16#6ADC;
   // GBK_TO_UNICODE[9350] := 16#99B3;
   // GBK_TO_UNICODE[9351] := 16#6ADD;
   // GBK_TO_UNICODE[9352] := 16#99B4;
   // GBK_TO_UNICODE[9353] := 16#6ADE;
   // GBK_TO_UNICODE[9354] := 16#99B5;
   // GBK_TO_UNICODE[9355] := 16#6ADF;
   // GBK_TO_UNICODE[9356] := 16#99B6;
   // GBK_TO_UNICODE[9357] := 16#6AE0;
   // GBK_TO_UNICODE[9358] := 16#99B7;
   // GBK_TO_UNICODE[9359] := 16#6AE1;
   // GBK_TO_UNICODE[9360] := 16#99B8;
   // GBK_TO_UNICODE[9361] := 16#6AE2;
   // GBK_TO_UNICODE[9362] := 16#99B9;
   // GBK_TO_UNICODE[9363] := 16#6AE3;
   // GBK_TO_UNICODE[9364] := 16#99BA;
   // GBK_TO_UNICODE[9365] := 16#6AE4;
   // GBK_TO_UNICODE[9366] := 16#99BB;
   // GBK_TO_UNICODE[9367] := 16#6AE5;
   // GBK_TO_UNICODE[9368] := 16#99BC;
   // GBK_TO_UNICODE[9369] := 16#6AE6;
   // GBK_TO_UNICODE[9370] := 16#99BD;
   // GBK_TO_UNICODE[9371] := 16#6AE7;
   // GBK_TO_UNICODE[9372] := 16#99BE;
   // GBK_TO_UNICODE[9373] := 16#6AE8;
   // GBK_TO_UNICODE[9374] := 16#99BF;
   // GBK_TO_UNICODE[9375] := 16#6AE9;
   // GBK_TO_UNICODE[9376] := 16#99C0;
   // GBK_TO_UNICODE[9377] := 16#6AEA;
   // GBK_TO_UNICODE[9378] := 16#99C1;
   // GBK_TO_UNICODE[9379] := 16#6AEB;
   // GBK_TO_UNICODE[9380] := 16#99C2;
   // GBK_TO_UNICODE[9381] := 16#6AEC;
   // GBK_TO_UNICODE[9382] := 16#99C3;
   // GBK_TO_UNICODE[9383] := 16#6AED;
   // GBK_TO_UNICODE[9384] := 16#99C4;
   // GBK_TO_UNICODE[9385] := 16#6AEE;
   // GBK_TO_UNICODE[9386] := 16#99C5;
   // GBK_TO_UNICODE[9387] := 16#6AEF;
   // GBK_TO_UNICODE[9388] := 16#99C6;
   // GBK_TO_UNICODE[9389] := 16#6AF0;
   // GBK_TO_UNICODE[9390] := 16#99C7;
   // GBK_TO_UNICODE[9391] := 16#6AF1;
   // GBK_TO_UNICODE[9392] := 16#99C8;
   // GBK_TO_UNICODE[9393] := 16#6AF2;
   // GBK_TO_UNICODE[9394] := 16#99C9;
   // GBK_TO_UNICODE[9395] := 16#6AF3;
   // GBK_TO_UNICODE[9396] := 16#99CA;
   // GBK_TO_UNICODE[9397] := 16#6AF4;
   // GBK_TO_UNICODE[9398] := 16#99CB;
   // GBK_TO_UNICODE[9399] := 16#6AF5;
   // GBK_TO_UNICODE[9400] := 16#99CC;
   // GBK_TO_UNICODE[9401] := 16#6AF6;
   // GBK_TO_UNICODE[9402] := 16#99CD;
   // GBK_TO_UNICODE[9403] := 16#6AF7;
   // GBK_TO_UNICODE[9404] := 16#99CE;
   // GBK_TO_UNICODE[9405] := 16#6AF8;
   // GBK_TO_UNICODE[9406] := 16#99CF;
   // GBK_TO_UNICODE[9407] := 16#6AF9;
   // GBK_TO_UNICODE[9408] := 16#99D0;
   // GBK_TO_UNICODE[9409] := 16#6AFA;
   // GBK_TO_UNICODE[9410] := 16#99D1;
   // GBK_TO_UNICODE[9411] := 16#6AFB;
   // GBK_TO_UNICODE[9412] := 16#99D2;
   // GBK_TO_UNICODE[9413] := 16#6AFC;
   // GBK_TO_UNICODE[9414] := 16#99D3;
   // GBK_TO_UNICODE[9415] := 16#6AFD;
   // GBK_TO_UNICODE[9416] := 16#99D4;
   // GBK_TO_UNICODE[9417] := 16#6AFE;
   // GBK_TO_UNICODE[9418] := 16#99D5;
   // GBK_TO_UNICODE[9419] := 16#6AFF;
   // GBK_TO_UNICODE[9420] := 16#99D6;
   // GBK_TO_UNICODE[9421] := 16#6B00;
   // GBK_TO_UNICODE[9422] := 16#99D7;
   // GBK_TO_UNICODE[9423] := 16#6B01;
   // GBK_TO_UNICODE[9424] := 16#99D8;
   // GBK_TO_UNICODE[9425] := 16#6B02;
   // GBK_TO_UNICODE[9426] := 16#99D9;
   // GBK_TO_UNICODE[9427] := 16#6B03;
   // GBK_TO_UNICODE[9428] := 16#99DA;
   // GBK_TO_UNICODE[9429] := 16#6B04;
   // GBK_TO_UNICODE[9430] := 16#99DB;
   // GBK_TO_UNICODE[9431] := 16#6B05;
   // GBK_TO_UNICODE[9432] := 16#99DC;
   // GBK_TO_UNICODE[9433] := 16#6B06;
   // GBK_TO_UNICODE[9434] := 16#99DD;
   // GBK_TO_UNICODE[9435] := 16#6B07;
   // GBK_TO_UNICODE[9436] := 16#99DE;
   // GBK_TO_UNICODE[9437] := 16#6B08;
   // GBK_TO_UNICODE[9438] := 16#99DF;
   // GBK_TO_UNICODE[9439] := 16#6B09;
   // GBK_TO_UNICODE[9440] := 16#99E0;
   // GBK_TO_UNICODE[9441] := 16#6B0A;
   // GBK_TO_UNICODE[9442] := 16#99E1;
   // GBK_TO_UNICODE[9443] := 16#6B0B;
   // GBK_TO_UNICODE[9444] := 16#99E2;
   // GBK_TO_UNICODE[9445] := 16#6B0C;
   // GBK_TO_UNICODE[9446] := 16#99E3;
   // GBK_TO_UNICODE[9447] := 16#6B0D;
   // GBK_TO_UNICODE[9448] := 16#99E4;
   // GBK_TO_UNICODE[9449] := 16#6B0E;
   // GBK_TO_UNICODE[9450] := 16#99E5;
   // GBK_TO_UNICODE[9451] := 16#6B0F;
   // GBK_TO_UNICODE[9452] := 16#99E6;
   // GBK_TO_UNICODE[9453] := 16#6B10;
   // GBK_TO_UNICODE[9454] := 16#99E7;
   // GBK_TO_UNICODE[9455] := 16#6B11;
   // GBK_TO_UNICODE[9456] := 16#99E8;
   // GBK_TO_UNICODE[9457] := 16#6B12;
   // GBK_TO_UNICODE[9458] := 16#99E9;
   // GBK_TO_UNICODE[9459] := 16#6B13;
   // GBK_TO_UNICODE[9460] := 16#99EA;
   // GBK_TO_UNICODE[9461] := 16#6B14;
   // GBK_TO_UNICODE[9462] := 16#99EB;
   // GBK_TO_UNICODE[9463] := 16#6B15;
   // GBK_TO_UNICODE[9464] := 16#99EC;
   // GBK_TO_UNICODE[9465] := 16#6B16;
   // GBK_TO_UNICODE[9466] := 16#99ED;
   // GBK_TO_UNICODE[9467] := 16#6B17;
   // GBK_TO_UNICODE[9468] := 16#99EE;
   // GBK_TO_UNICODE[9469] := 16#6B18;
   // GBK_TO_UNICODE[9470] := 16#99EF;
   // GBK_TO_UNICODE[9471] := 16#6B19;
   // GBK_TO_UNICODE[9472] := 16#99F0;
   // GBK_TO_UNICODE[9473] := 16#6B1A;
   // GBK_TO_UNICODE[9474] := 16#99F1;
   // GBK_TO_UNICODE[9475] := 16#6B1B;
   // GBK_TO_UNICODE[9476] := 16#99F2;
   // GBK_TO_UNICODE[9477] := 16#6B1C;
   // GBK_TO_UNICODE[9478] := 16#99F3;
   // GBK_TO_UNICODE[9479] := 16#6B1D;
   // GBK_TO_UNICODE[9480] := 16#99F4;
   // GBK_TO_UNICODE[9481] := 16#6B1E;
   // GBK_TO_UNICODE[9482] := 16#99F5;
   // GBK_TO_UNICODE[9483] := 16#6B1F;
   // GBK_TO_UNICODE[9484] := 16#99F6;
   // GBK_TO_UNICODE[9485] := 16#6B25;
   // GBK_TO_UNICODE[9486] := 16#99F7;
   // GBK_TO_UNICODE[9487] := 16#6B26;
   // GBK_TO_UNICODE[9488] := 16#99F8;
   // GBK_TO_UNICODE[9489] := 16#6B28;
   // GBK_TO_UNICODE[9490] := 16#99F9;
   // GBK_TO_UNICODE[9491] := 16#6B29;
   // GBK_TO_UNICODE[9492] := 16#99FA;
   // GBK_TO_UNICODE[9493] := 16#6B2A;
   // GBK_TO_UNICODE[9494] := 16#99FB;
   // GBK_TO_UNICODE[9495] := 16#6B2B;
   // GBK_TO_UNICODE[9496] := 16#99FC;
   // GBK_TO_UNICODE[9497] := 16#6B2C;
   // GBK_TO_UNICODE[9498] := 16#99FD;
   // GBK_TO_UNICODE[9499] := 16#6B2D;
   // GBK_TO_UNICODE[9500] := 16#99FE;
   // GBK_TO_UNICODE[9501] := 16#6B2E;
   // GBK_TO_UNICODE[9502] := 16#9A40;
   // GBK_TO_UNICODE[9503] := 16#6B2F;
   // GBK_TO_UNICODE[9504] := 16#9A41;
   // GBK_TO_UNICODE[9505] := 16#6B30;
   // GBK_TO_UNICODE[9506] := 16#9A42;
   // GBK_TO_UNICODE[9507] := 16#6B31;
   // GBK_TO_UNICODE[9508] := 16#9A43;
   // GBK_TO_UNICODE[9509] := 16#6B33;
   // GBK_TO_UNICODE[9510] := 16#9A44;
   // GBK_TO_UNICODE[9511] := 16#6B34;
   // GBK_TO_UNICODE[9512] := 16#9A45;
   // GBK_TO_UNICODE[9513] := 16#6B35;
   // GBK_TO_UNICODE[9514] := 16#9A46;
   // GBK_TO_UNICODE[9515] := 16#6B36;
   // GBK_TO_UNICODE[9516] := 16#9A47;
   // GBK_TO_UNICODE[9517] := 16#6B38;
   // GBK_TO_UNICODE[9518] := 16#9A48;
   // GBK_TO_UNICODE[9519] := 16#6B3B;
   // GBK_TO_UNICODE[9520] := 16#9A49;
   // GBK_TO_UNICODE[9521] := 16#6B3C;
   // GBK_TO_UNICODE[9522] := 16#9A4A;
   // GBK_TO_UNICODE[9523] := 16#6B3D;
   // GBK_TO_UNICODE[9524] := 16#9A4B;
   // GBK_TO_UNICODE[9525] := 16#6B3F;
   // GBK_TO_UNICODE[9526] := 16#9A4C;
   // GBK_TO_UNICODE[9527] := 16#6B40;
   // GBK_TO_UNICODE[9528] := 16#9A4D;
   // GBK_TO_UNICODE[9529] := 16#6B41;
   // GBK_TO_UNICODE[9530] := 16#9A4E;
   // GBK_TO_UNICODE[9531] := 16#6B42;
   // GBK_TO_UNICODE[9532] := 16#9A4F;
   // GBK_TO_UNICODE[9533] := 16#6B44;
   // GBK_TO_UNICODE[9534] := 16#9A50;
   // GBK_TO_UNICODE[9535] := 16#6B45;
   // GBK_TO_UNICODE[9536] := 16#9A51;
   // GBK_TO_UNICODE[9537] := 16#6B48;
   // GBK_TO_UNICODE[9538] := 16#9A52;
   // GBK_TO_UNICODE[9539] := 16#6B4A;
   // GBK_TO_UNICODE[9540] := 16#9A53;
   // GBK_TO_UNICODE[9541] := 16#6B4B;
   // GBK_TO_UNICODE[9542] := 16#9A54;
   // GBK_TO_UNICODE[9543] := 16#6B4D;
   // GBK_TO_UNICODE[9544] := 16#9A55;
   // GBK_TO_UNICODE[9545] := 16#6B4E;
   // GBK_TO_UNICODE[9546] := 16#9A56;
   // GBK_TO_UNICODE[9547] := 16#6B4F;
   // GBK_TO_UNICODE[9548] := 16#9A57;
   // GBK_TO_UNICODE[9549] := 16#6B50;
   // GBK_TO_UNICODE[9550] := 16#9A58;
   // GBK_TO_UNICODE[9551] := 16#6B51;
   // GBK_TO_UNICODE[9552] := 16#9A59;
   // GBK_TO_UNICODE[9553] := 16#6B52;
   // GBK_TO_UNICODE[9554] := 16#9A5A;
   // GBK_TO_UNICODE[9555] := 16#6B53;
   // GBK_TO_UNICODE[9556] := 16#9A5B;
